KUKA KRL program: MyProgram_212().src

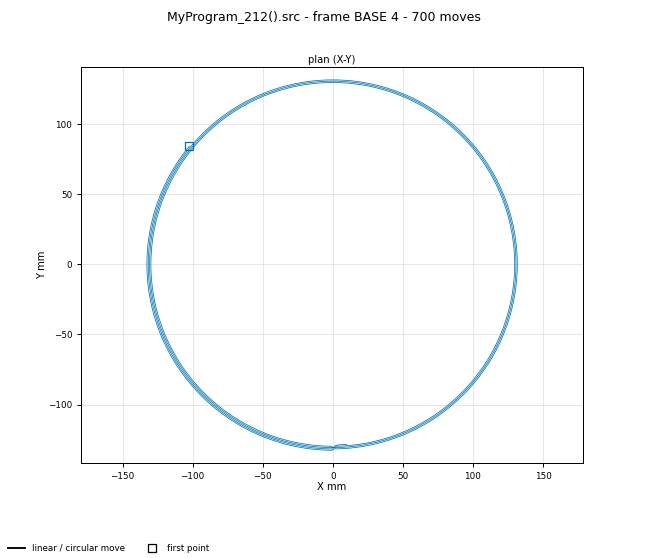
[picture p0: tool path of MyProgram_212().src in frame BASE 4, 700 of 700 moves have a stored position in this frame; points joined in program order, loops and branches not executed]
&ACCESS RVP
&REL 1
&PARAM TEMPLATE = C:\KRC\Roboter\Template\vorgabe
&PARAM EDITMASK = *
DEF MyProgram_212()
; ---- Setting reference (Base) ----
$BASE = BASE_DATA[4]

; --------------------------
; ---- Setting tool (TCP) ----
$TOOL = TOOL_DATA[3]
; --------------------------

$VEL.CP = VEL_APROX_PRINT
Startdeposition()
$VEL.CP = VEL_PRINT
LIN {X -102.2759,Y 84.4274,Z 150,A 136.9354,B 24.9526,C -1.5903,E1 24.8761,E2 309.4983} C_DIS
LIN {X -104.8003,Y 81.2724,Z 150,A 138.873,B 24.9523,C -1.5949,E1 24.8727,E2 307.5405} C_DIS
LIN {X -107.3516,Y 77.8713,Z 150,A 140.7222,B 24.9526,C -1.5904,E1 24.8697,E2 305.6931} C_DIS
LIN {X -109.8219,Y 74.3469,Z 150,A 142.615,B 24.9528,C -1.5868,E1 24.8667,E2 303.7996} C_DIS
LIN {X -112.2899,Y 70.5646,Z 150,A 144.5743,B 24.9531,C -1.5815,E1 24.8637,E2 301.8428} C_DIS
LIN {X -114.4855,Y 66.9437,Z 150,A 146.4163,B 24.9534,C -1.5768,E1 24.8611,E2 300.0027} C_DIS
LIN {X -116.5889,Y 63.2096,Z 150,A 148.3143,B 24.9536,C -1.5735,E1 24.8585,E2 298.1025} C_DIS
LIN {X -118.1366,Y 60.2624,Z 150,A 149.6641,B 24.9541,C -1.5649,E1 24.8568,E2 296.7661} C_DIS
LIN {X -120.6399,Y 55.0837,Z 150,A 152.138,B 24.9546,C -1.5567,E1 24.8539,E2 294.2982} C_DIS
LIN {X -122.2455,Y 51.4194,Z 150,A 153.8562,B 24.9549,C -1.5508,E1 24.852,E2 292.5846} C_DIS
LIN {X -123.5059,Y 48.3134,Z 150,A 155.3546,B 24.9551,C -1.5487,E1 24.8504,E2 291.0827} C_DIS
LIN {X -124.7525,Y 44.9959,Z 150,A 156.841,B 24.9555,C -1.5417,E1 24.849,E2 289.6046} C_DIS
LIN {X -125.7894,Y 42.0105,Z 150,A 158.2756,B 24.9555,C -1.5407,E1 24.8477,E2 288.1643} C_DIS
LIN {X -126.918,Y 38.468,Z 150,A 159.9592,B 24.9556,C -1.5393,E1 24.8463,E2 286.4744} C_DIS
LIN {X -128.0963,Y 34.3396,Z 150,A 161.7856,B 24.956,C -1.5319,E1 24.845,E2 284.655} C_DIS
LIN {X -129.0879,Y 30.4082,Z 150,A 163.4654,B 24.9566,C -1.5227,E1 24.8439,E2 282.9873} C_DIS
LIN {X -130.1134,Y 25.671,Z 150,A 165.7274,B 24.9565,C -1.5239,E1 24.8426,E2 280.709} C_DIS
LIN {X -130.8013,Y 21.8842,Z 150,A 167.3023,B 24.957,C -1.5143,E1 24.8418,E2 279.1478} C_DIS
LIN {X -131.3985,Y 17.9691,Z 150,A 169.2633,B 24.9567,C -1.5207,E1 24.841,E2 277.1597} C_DIS
LIN {X -131.9911,Y 12.8966,Z 150,A 171.2061,B 24.9578,C -1.5007,E1 24.8405,E2 275.2531} C_DIS
LIN {X -132.2828,Y 9.4461,Z 150,A 172.7501,B 24.958,C -1.498,E1 24.8401,E2 273.7061} C_DIS
LIN {X -132.5132,Y 5.3118,Z 150,A 174.5305,B 24.9583,C -1.4917,E1 24.8399,E2 271.93} C_DIS
LIN {X -132.6019,Y 2.1638,Z 150,A 175.9323,B 24.9585,C -1.4892,E1 24.8398,E2 270.5258} C_DIS
LIN {X -132.6079,Y -1.8067,Z 150,A 177.6767,B 24.9587,C -1.4849,E1 24.8398,E2 268.781} C_DIS
LIN {X -132.4992,Y -5.6705,Z 150,A 179.3978,B 24.9589,C -1.4819,E1 24.84,E2 267.0568} C_DIS
LIN {X -132.2762,Y -9.5365,Z 150,A -178.6096,B 24.9583,C -1.492,E1 24.8404,E2 265.0281} C_DIS
LIN {X -131.9496,Y -13.3288,Z 150,A -177.2383,B 24.9593,C -1.4733,E1 24.8408,E2 263.6932} C_DIS
LIN {X -131.5115,Y -17.1072,Z 150,A -175.6535,B 24.9598,C -1.4651,E1 24.8413,E2 262.1183} C_DIS
LIN {X -130.9322,Y -21.0996,Z 150,A -173.9674,B 24.9602,C -1.4567,E1 24.842,E2 260.4423} C_DIS
LIN {X -130.2084,Y -25.1739,Z 150,A -172.0506,B 24.9602,C -1.4573,E1 24.843,E2 258.5128} C_DIS
LIN {X -129.3647,Y -29.2021,Z 150,A -170.3174,B 24.9606,C -1.4494,E1 24.844,E2 256.7881} C_DIS
LIN {X -128.5771,Y -32.4932,Z 150,A -168.8558,B 24.9609,C -1.4448,E1 24.845,E2 255.3289} C_DIS
LIN {X -127.6515,Y -35.9585,Z 150,A -167.2711,B 24.9611,C -1.4417,E1 24.8461,E2 253.7426} C_DIS
LIN {X -126.4549,Y -39.9645,Z 150,A -165.4673,B 24.9614,C -1.436,E1 24.8476,E2 251.9419} C_DIS
LIN {X -125.4607,Y -42.9847,Z 150,A -164.0858,B 24.9616,C -1.4321,E1 24.8489,E2 250.5617} C_DIS
LIN {X -124.3657,Y -46.0568,Z 150,A -162.3318,B 24.9609,C -1.4448,E1 24.8506,E2 248.7676} C_DIS
LIN {X -123.1055,Y -49.3248,Z 150,A -161.0063,B 24.9616,C -1.431,E1 24.8519,E2 247.4675} C_DIS
LIN {X -121.3813,Y -53.4321,Z 150,A -159.1275,B 24.9621,C -1.4231,E1 24.854,E2 245.5972} C_DIS
LIN {X -119.781,Y -56.9243,Z 150,A -157.5495,B 24.9625,C -1.4143,E1 24.8558,E2 244.0315} C_DIS
LIN {X -118.2712,Y -59.998,Z 150,A -156.0681,B 24.9627,C -1.4102,E1 24.8577,E2 242.5519} C_DIS
LIN {X -116.633,Y -63.1286,Z 150,A -154.4098,B 24.9627,C -1.4123,E1 24.8599,E2 240.8797} C_DIS
LIN {X -114.4561,Y -66.9937,Z 150,A -152.521,B 24.963,C -1.4057,E1 24.8625,E2 238.997} C_DIS
LIN {X -112.2679,Y -70.5995,Z 150,A -150.6806,B 24.9632,C -1.4017,E1 24.8652,E2 237.1567} C_DIS
LIN {X -109.8561,Y -74.2964,Z 150,A -149.0433,B 24.9642,C -1.3834,E1 24.8677,E2 235.5548} C_DIS
LIN {X -108.2088,Y -76.6762,Z 150,A -147.5106,B 24.9636,C -1.3941,E1 24.8702,E2 233.9891} C_DIS
LIN {X -105.6102,Y -80.2182,Z 150,A -145.571,B 24.9637,C -1.3914,E1 24.8734,E2 232.0466} C_DIS
LIN {X -102.8564,Y -83.7194,Z 150,A -143.6381,B 24.964,C -1.3871,E1 24.8768,E2 230.1148} C_DIS
LIN {X -99.9263,Y -87.1954,Z 150,A -141.6922,B 24.9642,C -1.3816,E1 24.8803,E2 228.1732} C_DIS
LIN {X -96.9225,Y -90.5228,Z 150,A -139.7451,B 24.9644,C -1.3777,E1 24.884,E2 226.2267} C_DIS
LIN {X -93.8055,Y -93.7496,Z 150,A -137.7952,B 24.9646,C -1.374,E1 24.8878,E2 224.2774} C_DIS
LIN {X -90.7475,Y -96.7126,Z 150,A -135.9208,B 24.9647,C -1.3718,E1 24.8916,E2 222.4003} C_DIS
LIN {X -87.5016,Y -99.6591,Z 150,A -134.0241,B 24.9649,C -1.3681,E1 24.8956,E2 220.5048} C_DIS
LIN {X -84.1587,Y -102.4974,Z 150,A -132.1382,B 24.9651,C -1.364,E1 24.8996,E2 218.6215} C_DIS
LIN {X -80.768,Y -105.1898,Z 150,A -130.2526,B 24.9653,C -1.3613,E1 24.9038,E2 216.7355} C_DIS
LIN {X -77.1748,Y -107.8534,Z 150,A -128.3209,B 24.9655,C -1.3579,E1 24.9081,E2 214.8051} C_DIS
LIN {X -73.3393,Y -110.4979,Z 150,A -126.2967,B 24.9656,C -1.3551,E1 24.9128,E2 212.7807} C_DIS
LIN {X -69.7226,Y -112.8151,Z 150,A -124.4068,B 24.9656,C -1.3539,E1 24.9173,E2 210.8876} C_DIS
LIN {X -65.5266,Y -115.3023,Z 150,A -122.009,B 24.9651,C -1.3657,E1 24.9232,E2 208.4548} C_DIS
LIN {X -62.1909,Y -117.1343,Z 150,A -120.678,B 24.966,C -1.3475,E1 24.9264,E2 207.1634} C_DIS
LIN {X -58.8187,Y -118.8621,Z 150,A -119.1574,B 24.9664,C -1.3395,E1 24.9301,E2 205.6577} C_DIS
LIN {X -55.5234,Y -120.4366,Z 150,A -117.5891,B 24.9665,C -1.3371,E1 24.9341,E2 204.0912} C_DIS
LIN {X -52.7823,Y -121.6629,Z 150,A -116.3412,B 24.9667,C -1.3331,E1 24.9373,E2 202.8497} C_DIS
LIN {X -49.8052,Y -122.9118,Z 150,A -114.8731,B 24.9666,C -1.3354,E1 24.9411,E2 201.3728} C_DIS
LIN {X -46.6232,Y -124.1536,Z 150,A -113.396,B 24.9666,C -1.334,E1 24.9449,E2 199.8959} C_DIS
LIN {X -43.6406,Y -125.2333,Z 150,A -111.9841,B 24.9666,C -1.3349,E1 24.9486,E2 198.479} C_DIS
LIN {X -40.3714,Y -126.3249,Z 150,A -110.5705,B 24.9669,C -1.3299,E1 24.9524,E2 197.0749} C_DIS
LIN {X -36.267,Y -127.5652,Z 150,A -108.6068,B 24.9667,C -1.3343,E1 24.9577,E2 195.0975} C_DIS
LIN {X -32.2664,Y -128.6346,Z 150,A -106.7479,B 24.9665,C -1.3368,E1 24.9627,E2 193.2298} C_DIS
LIN {X -28.2908,Y -129.567,Z 150,A -105.0688,B 24.9668,C -1.3315,E1 24.9673,E2 191.5612} C_DIS
LIN {X -24.1984,Y -130.3949,Z 150,A -103.1867,B 24.9666,C -1.3348,E1 24.9724,E2 189.6691} C_DIS
LIN {X -20.4691,Y -131.0303,Z 150,A -101.6331,B 24.9669,C -1.3302,E1 24.9767,E2 188.1251} C_DIS
LIN {X -16.8245,Y -131.5485,Z 150,A -99.9382,B 24.9666,C -1.3353,E1 24.9814,E2 186.4168} C_DIS
LIN {X -13.0464,Y -131.9767,Z 150,A -98.3401,B 24.9667,C -1.3328,E1 24.9859,E2 184.8237} C_DIS
LIN {X -8.7557,Y -132.3315,Z 150,A -96.4662,B 24.9667,C -1.3334,E1 24.9911,E2 182.9475} C_DIS
LIN {X -4.8645,Y -132.5306,Z 150,A -94.7842,B 24.9667,C -1.3335,E1 24.9958,E2 181.2649} C_DIS
LIN {X -0.6926,Y -132.6178,Z 150,A -93.0498,B 24.9669,C -1.3303,E1 25.0006,E2 179.5381} C_DIS
LIN {X -0.6926,Y -132.6178,Z 150,A -93.0498,B 24.9669,C -1.3303,E1 25.0006,E2 179.5381} C_DIS
Enddeposition()
LIN {X 0.9332,Y -131.667,Z 150,A -92.4211,B 24.2531,C -1.1938,E1 24.2824,E2 179.1428} C_DIS
Startdeposition()
$VEL.CP = VEL_PRINT
LIN {X -0.8148,Y -131.6701,Z 150,A -93.6093,B 24.2541,C -1.1721,E1 24.279,E2 180.3838} C_DIS
LIN {X -4.9682,Y -131.5789,Z 150,A -95.3944,B 24.2541,C -1.173,E1 24.274,E2 182.1669} C_DIS
LIN {X -8.4532,Y -131.4014,Z 150,A -96.8971,B 24.2541,C -1.1737,E1 24.2698,E2 183.6683} C_DIS
LIN {X -11.7251,Y -131.151,Z 150,A -98.299,B 24.2541,C -1.1751,E1 24.2659,E2 185.0676} C_DIS
LIN {X -15.4301,Y -130.7653,Z 150,A -99.9452,B 24.2541,C -1.174,E1 24.2613,E2 186.7174} C_DIS
LIN {X -18.6917,Y -130.339,Z 150,A -101.3801,B 24.2541,C -1.1742,E1 24.2574,E2 188.1531} C_DIS
LIN {X -22.0826,Y -129.8081,Z 150,A -102.8712,B 24.2541,C -1.1747,E1 24.2532,E2 189.6442} C_DIS
LIN {X -25.4894,Y -129.184,Z 150,A -104.363,B 24.254,C -1.1761,E1 24.2492,E2 191.1344} C_DIS
LIN {X -27.9438,Y -128.6731,Z 150,A -105.4714,B 24.254,C -1.1757,E1 24.2461,E2 192.245} C_DIS
LIN {X -31.6236,Y -127.8208,Z 150,A -107.1045,B 24.254,C -1.1771,E1 24.2417,E2 193.877} C_DIS
LIN {X -34.5863,Y -127.0505,Z 150,A -108.4405,B 24.2539,C -1.1777,E1 24.2381,E2 195.2135} C_DIS
LIN {X -37.6577,Y -126.1742,Z 150,A -109.8155,B 24.2539,C -1.1794,E1 24.2344,E2 196.5867} C_DIS
LIN {X -40.1695,Y -125.3953,Z 150,A -110.9923,B 24.2539,C -1.1788,E1 24.2313,E2 197.7674} C_DIS
LIN {X -43.3579,Y -124.329,Z 150,A -112.4851,B 24.2539,C -1.1785,E1 24.2273,E2 199.2636} C_DIS
LIN {X -46.6138,Y -123.1459,Z 150,A -113.9587,B 24.2537,C -1.1816,E1 24.2235,E2 200.733} C_DIS
LIN {X -49.5228,Y -122.0046,Z 150,A -115.3569,B 24.2537,C -1.1811,E1 24.2198,E2 202.1355} C_DIS
LIN {X -52.7628,Y -120.6397,Z 150,A -116.8575,B 24.2536,C -1.1842,E1 24.216,E2 203.6323} C_DIS
LIN {X -56.0138,Y -119.1665,Z 150,A -118.4198,B 24.2536,C -1.1855,E1 24.212,E2 205.1953} C_DIS
LIN {X -58.9958,Y -117.7187,Z 150,A -119.9107,B 24.2536,C -1.185,E1 24.2083,E2 206.6915} C_DIS
LIN {X -62.6349,Y -115.8233,Z 150,A -121.6598,B 24.2534,C -1.1891,E1 24.204,E2 208.4356} C_DIS
LIN {X -65.5557,Y -114.1955,Z 150,A -123.2346,B 24.2535,C -1.1854,E1 24.2001,E2 210.0242} C_DIS
LIN {X -69.2621,Y -111.9863,Z 150,A -125.1463,B 24.2535,C -1.1866,E1 24.1955,E2 211.9391} C_DIS
LIN {X -72.6874,Y -109.7938,Z 150,A -126.8783,B 24.2533,C -1.1912,E1 24.1915,E2 213.6656} C_DIS
LIN {X -76.2415,Y -107.3566,Z 150,A -128.6594,B 24.2529,C -1.1989,E1 24.1874,E2 215.4341} C_DIS
LIN {X -79.3271,Y -105.0963,Z 150,A -130.393,B 24.2529,C -1.1986,E1 24.1835,E2 217.175} C_DIS
LIN {X -82.6146,Y -102.5322,Z 150,A -132.2309,B 24.2529,C -1.2008,E1 24.1795,E2 219.0145} C_DIS
LIN {X -85.8963,Y -99.7991,Z 150,A -134.0859,B 24.2526,C -1.2046,E1 24.1756,E2 220.8676} C_DIS
LIN {X -88.9982,Y -97.0431,Z 150,A -135.9311,B 24.2526,C -1.2064,E1 24.1717,E2 222.7161} C_DIS
LIN {X -91.8951,Y -94.3054,Z 150,A -137.5823,B 24.2522,C -1.214,E1 24.1684,E2 224.3558} C_DIS
LIN {X -94.2367,Y -91.9651,Z 150,A -139.1194,B 24.2522,C -1.2125,E1 24.1654,E2 225.9031} C_DIS
LIN {X -97.2286,Y -88.7965,Z 150,A -140.9291,B 24.2519,C -1.2209,E1 24.162,E2 227.7007} C_DIS
LIN {X -99.4528,Y -86.2977,Z 150,A -142.3879,B 24.2517,C -1.2241,E1 24.1593,E2 229.1584} C_DIS
LIN {X -101.8838,Y -83.413,Z 150,A -144.1386,B 24.2517,C -1.2229,E1 24.1561,E2 230.9203} C_DIS
LIN {X -104.5752,Y -80.0129,Z 150,A -146.0156,B 24.2515,C -1.228,E1 24.1529,E2 232.7941} C_DIS
LIN {X -107.0701,Y -76.6422,Z 150,A -147.8508,B 24.2513,C -1.2321,E1 24.1499,E2 234.6284} C_DIS
LIN {X -109.4269,Y -73.2379,Z 150,A -149.6804,B 24.2512,C -1.2355,E1 24.147,E2 236.4593} C_DIS
LIN {X -111.5415,Y -69.9761,Z 150,A -151.3797,B 24.251,C -1.2396,E1 24.1445,E2 238.1574} C_DIS
LIN {X -113.7761,Y -66.2809,Z 150,A -153.3185,B 24.2509,C -1.2419,E1 24.1417,E2 240.1008} C_DIS
LIN {X -115.7952,Y -62.6871,Z 150,A -155.1261,B 24.2507,C -1.2462,E1 24.1393,E2 241.9078} C_DIS
LIN {X -117.5957,Y -59.2374,Z 150,A -156.678,B 24.2501,C -1.2575,E1 24.1373,E2 243.4405} C_DIS
LIN {X -118.9999,Y -56.3627,Z 150,A -158.0771,B 24.2499,C -1.2612,E1 24.1356,E2 244.8385} C_DIS
LIN {X -120.5329,Y -53.0096,Z 150,A -159.6961,B 24.2498,C -1.2651,E1 24.1338,E2 246.457} C_DIS
LIN {X -121.8177,Y -49.9865,Z 150,A -161.133,B 24.2496,C -1.269,E1 24.1322,E2 247.8927} C_DIS
LIN {X -123.0209,Y -46.9474,Z 150,A -162.5629,B 24.2494,C -1.2729,E1 24.1308,E2 249.3214} C_DIS
LIN {X -123.9898,Y -44.3194,Z 150,A -163.8263,B 24.2493,C -1.2745,E1 24.1296,E2 250.5881} C_DIS
LIN {X -125.0082,Y -41.3591,Z 150,A -165.1834,B 24.2491,C -1.2789,E1 24.1284,E2 251.9425} C_DIS
LIN {X -126.0115,Y -38.1942,Z 150,A -166.5921,B 24.2488,C -1.285,E1 24.1272,E2 253.3447} C_DIS
LIN {X -126.826,Y -35.3942,Z 150,A -167.883,B 24.2486,C -1.2879,E1 24.1262,E2 254.6362} C_DIS
LIN {X -127.6413,Y -32.3308,Z 150,A -169.2828,B 24.2485,C -1.2912,E1 24.1252,E2 256.0363} C_DIS
LIN {X -128.4131,Y -29.1152,Z 150,A -170.728,B 24.2482,C -1.2955,E1 24.1243,E2 257.4798} C_DIS
LIN {X -129.0911,Y -25.9459,Z 150,A -172.1707,B 24.2481,C -1.2984,E1 24.1235,E2 258.924} C_DIS
LIN {X -129.7497,Y -22.4326,Z 150,A -173.7009,B 24.2478,C -1.3045,E1 24.1227,E2 260.4487} C_DIS
LIN {X -130.2397,Y -19.3862,Z 150,A -175.0507,B 24.2476,C -1.3085,E1 24.1222,E2 261.7971} C_DIS
LIN {X -130.6553,Y -16.3526,Z 150,A -176.3905,B 24.2474,C -1.3124,E1 24.1217,E2 263.1355} C_DIS
LIN {X -130.9862,Y -13.4413,Z 150,A -177.6717,B 24.2472,C -1.3163,E1 24.1213,E2 264.4153} C_DIS
LIN {X -131.2685,Y -10.3335,Z 150,A -179.0367,B 24.247,C -1.3203,E1 24.121,E2 265.7788} C_DIS
LIN {X -131.4334,Y -7.9342,Z 150,A 179.8473,B 24.247,C -1.3206,E1 24.1208,E2 266.9011} C_DIS
LIN {X -131.5972,Y -4.4983,Z 150,A 178.404,B 24.2466,C -1.3279,E1 24.1206,E2 268.3355} C_DIS
LIN {X -131.6648,Y -1.5621,Z 150,A 177.1632,B 24.2463,C -1.3338,E1 24.1206,E2 269.5697} C_DIS
LIN {X -131.6678,Y 1.287,Z 150,A 175.8565,B 24.2463,C -1.3348,E1 24.1206,E2 270.882} C_DIS
LIN {X -131.5674,Y 5.2629,Z 150,A 174.0649,B 24.2461,C -1.3377,E1 24.1206,E2 272.6777} C_DIS
LIN {X -131.3775,Y 8.8404,Z 150,A 172.5524,B 24.2457,C -1.3449,E1 24.1209,E2 274.182} C_DIS
LIN {X -131.151,Y 11.7251,Z 150,A 171.279,B 24.2455,C -1.3484,E1 24.1212,E2 275.4547} C_DIS
LIN {X -130.836,Y 14.837,Z 150,A 169.9092,B 24.2453,C -1.3524,E1 24.1217,E2 276.8231} C_DIS
LIN {X -130.4708,Y 17.76,Z 150,A 168.6347,B 24.2451,C -1.3569,E1 24.1221,E2 278.0944} C_DIS
LIN {X -130.0208,Y 20.7999,Z 150,A 167.2633,B 24.2449,C -1.3597,E1 24.1227,E2 279.4673} C_DIS
LIN {X -129.4958,Y 23.8514,Z 150,A 165.9042,B 24.2447,C -1.3636,E1 24.1234,E2 280.8253} C_DIS
LIN {X -128.9359,Y 26.7086,Z 150,A 164.6144,B 24.2446,C -1.3667,E1 24.1241,E2 282.1154} C_DIS
LIN {X -128.2739,Y 29.725,Z 150,A 163.2857,B 24.2443,C -1.3717,E1 24.1249,E2 283.4399} C_DIS
LIN {X -127.4587,Y 33.0503,Z 150,A 161.771,B 24.2441,C -1.3754,E1 24.1259,E2 284.9548} C_DIS
LIN {X -126.7683,Y 35.6006,Z 150,A 160.5988,B 24.244,C -1.3781,E1 24.1268,E2 286.1274} C_DIS
LIN {X -125.8001,Y 38.8849,Z 150,A 159.1337,B 24.2437,C -1.3839,E1 24.128,E2 287.5869} C_DIS
LIN {X -124.8443,Y 41.8511,Z 150,A 157.7294,B 24.2435,C -1.386,E1 24.1292,E2 288.9944} C_DIS
LIN {X -123.7058,Y 45.1071,Z 150,A 156.251,B 24.2432,C -1.3918,E1 24.1306,E2 290.4673} C_DIS
LIN {X -122.5781,Y 48.0866,Z 150,A 154.8065,B 24.2432,C -1.3935,E1 24.132,E2 291.9161} C_DIS
LIN {X -121.3681,Y 51.0632,Z 150,A 153.3887,B 24.243,C -1.3969,E1 24.1335,E2 293.3336} C_DIS
LIN {X -119.9077,Y 54.4074,Z 150,A 151.8353,B 24.2426,C -1.4033,E1 24.1353,E2 294.8801} C_DIS
LIN {X -118.4528,Y 57.5078,Z 150,A 150.3202,B 24.2424,C -1.4067,E1 24.1371,E2 296.3955} C_DIS
LIN {X -116.9645,Y 60.4774,Z 150,A 148.8639,B 24.2422,C -1.4106,E1 24.1389,E2 297.8504} C_DIS
LIN {X -115.4701,Y 63.2831,Z 150,A 147.3765,B 24.2422,C -1.4099,E1 24.1409,E2 299.3476} C_DIS
LIN {X -113.3517,Y 67.0041,Z 150,A 145.5412,B 24.2419,C -1.4166,E1 24.1435,E2 301.1762} C_DIS
LIN {X -111.1242,Y 70.6373,Z 150,A 143.7265,B 24.2415,C -1.4238,E1 24.1462,E2 302.9829} C_DIS
LIN {X -109.312,Y 73.4102,Z 150,A 142.2732,B 24.2413,C -1.4273,E1 24.1484,E2 304.4352} C_DIS
LIN {X -107.047,Y 76.6745,Z 150,A 140.4571,B 24.2413,C -1.4281,E1 24.1513,E2 306.2584} C_DIS
LIN {X -104.3697,Y 80.2816,Z 150,A 138.5679,B 24.2408,C -1.4365,E1 24.1545,E2 308.1366} C_DIS
LIN {X -102.226,Y 82.9943,Z 150,A 137.0243,B 24.2407,C -1.4387,E1 24.1572,E2 309.6823} C_DIS
LIN {X -99.5321,Y 86.2063,Z 150,A 135.2124,B 24.2404,C -1.4441,E1 24.1605,E2 311.4896} C_DIS
LIN {X -97.2692,Y 88.7516,Z 150,A 133.7284,B 24.2401,C -1.4478,E1 24.1632,E2 312.9714} C_DIS
LIN {X -94.9399,Y 91.2391,Z 150,A 132.2136,B 24.2401,C -1.45,E1 24.1661,E2 314.4875} C_DIS
LIN {X -92.0249,Y 94.178,Z 150,A 130.3391,B 24.24,C -1.451,E1 24.1699,E2 316.3677} C_DIS
LIN {X -88.7965,Y 97.2286,Z 150,A 128.4899,B 24.2395,C -1.4595,E1 24.1736,E2 318.204} C_DIS
LIN {X -86.2977,Y 99.4528,Z 150,A 127.021,B 24.2393,C -1.4622,E1 24.1767,E2 319.6722} C_DIS
LIN {X -83.6525,Y 101.6881,Z 150,A 125.4423,B 24.2393,C -1.4622,E1 24.1801,E2 321.257} C_DIS
LIN {X -80.3295,Y 104.333,Z 150,A 123.6507,B 24.239,C -1.4689,E1 24.184,E2 323.0393} C_DIS
LIN {X -77.6643,Y 106.3317,Z 150,A 122.1885,B 24.2388,C -1.4713,E1 24.1873,E2 324.5008} C_DIS
LIN {X -74.8561,Y 108.3271,Z 150,A 120.5702,B 24.239,C -1.4688,E1 24.191,E2 326.131} C_DIS
LIN {X -71.3969,Y 110.6374,Z 150,A 118.7929,B 24.2387,C -1.4739,E1 24.1952,E2 327.9019} C_DIS
LIN {X -67.8273,Y 112.861,Z 150,A 117.0305,B 24.2383,C -1.4805,E1 24.1993,E2 329.6539} C_DIS
LIN {X -64.4639,Y 114.8148,Z 150,A 115.2856,B 24.2383,C -1.4811,E1 24.2036,E2 331.4027} C_DIS
LIN {X -60.7251,Y 116.8344,Z 150,A 113.4927,B 24.2379,C -1.4869,E1 24.208,E2 333.1866} C_DIS
LIN {X -57.6492,Y 118.383,Z 150,A 111.9816,B 24.2379,C -1.4887,E1 24.2117,E2 334.6973} C_DIS
LIN {X -54.6208,Y 119.8106,Z 150,A 110.5189,B 24.2377,C -1.4907,E1 24.2154,E2 336.1589} C_DIS
LIN {X -51.6849,Y 121.1057,Z 150,A 109.114,B 24.2377,C -1.4923,E1 24.219,E2 337.5632} C_DIS
LIN {X -49.0101,Y 122.2113,Z 150,A 107.8485,B 24.2375,C -1.4938,E1 24.2223,E2 338.8279} C_DIS
LIN {X -45.8227,Y 123.4422,Z 150,A 106.3368,B 24.2375,C -1.4946,E1 24.2263,E2 340.3409} C_DIS
LIN {X -42.3661,Y 124.6728,Z 150,A 104.7722,B 24.2373,C -1.4981,E1 24.2304,E2 341.9002} C_DIS
LIN {X -39.4102,Y 125.6379,Z 150,A 103.4268,B 24.2372,C -1.5001,E1 24.2339,E2 343.2433} C_DIS
LIN {X -36.4873,Y 126.5169,Z 150,A 102.0875,B 24.2372,C -1.5011,E1 24.2375,E2 344.5825} C_DIS
LIN {X -33.4291,Y 127.3591,Z 150,A 100.6904,B 24.2371,C -1.5017,E1 24.2413,E2 345.9803} C_DIS
LIN {X -30.1974,Y 128.1646,Z 150,A 99.2568,B 24.2369,C -1.5038,E1 24.2452,E2 347.4108} C_DIS
LIN {X -27.4225,Y 128.7856,Z 150,A 97.9934,B 24.2369,C -1.5037,E1 24.2486,E2 348.6762} C_DIS
LIN {X -24.0686,Y 129.4556,Z 150,A 96.5273,B 24.2369,C -1.5059,E1 24.2526,E2 350.1384} C_DIS
LIN {X -21.0163,Y 129.986,Z 150,A 95.1792,B 24.2368,C -1.5069,E1 24.2564,E2 351.4855} C_DIS
LIN {X -18.3702,Y 130.3849,Z 150,A 93.9694,B 24.2368,C -1.5055,E1 24.2597,E2 352.6998} C_DIS
LIN {X -14.0764,Y 130.9179,Z 150,A 92.0983,B 24.2368,C -1.5071,E1 24.2649,E2 354.5681} C_DIS
LIN {X -10.8669,Y 131.2235,Z 150,A 90.6889,B 24.2368,C -1.5075,E1 24.2688,E2 355.9774} C_DIS
LIN {X -7.4582,Y 131.4627,Z 150,A 89.2712,B 24.2365,C -1.5114,E1 24.2727,E2 357.386} C_DIS
LIN {X -2.9226,Y 131.6422,Z 150,A 87.1562,B 24.2369,C -1.5052,E1 24.2787,E2 359.5166} C_DIS
LIN {X 0.7468,Y 131.6705,Z 150,A 85.6682,B 24.2365,C -1.5108,E1 24.2828,E2 360.9907} C_DIS
LIN {X 3.7909,Y 131.6181,Z 150,A 84.3302,B 24.2365,C -1.5103,E1 24.2865,E2 362.3297} C_DIS
LIN {X 7.2472,Y 131.4745,Z 150,A 82.8404,B 24.2365,C -1.5111,E1 24.2907,E2 363.8171} C_DIS
LIN {X 10.3335,Y 131.2685,Z 150,A 81.3369,B 24.237,C -1.5033,E1 24.2949,E2 365.3388} C_DIS
LIN {X 13.9989,Y 130.9262,Z 150,A 79.8614,B 24.2366,C -1.5093,E1 24.299,E2 366.7987} C_DIS
LIN {X 17.2091,Y 130.543,Z 150,A 78.4643,B 24.2366,C -1.5095,E1 24.3028,E2 368.1942} C_DIS
LIN {X 20.7999,Y 130.0208,Z 150,A 76.8983,B 24.2366,C -1.5096,E1 24.3072,E2 369.7585} C_DIS
LIN {X 23.8514,Y 129.4958,Z 150,A 75.5742,B 24.2366,C -1.5102,E1 24.3108,E2 371.0795} C_DIS
LIN {X 26.6183,Y 128.9542,Z 150,A 74.2994,B 24.2367,C -1.5073,E1 24.3143,E2 372.3598} C_DIS
LIN {X 30.0883,Y 128.1909,Z 150,A 72.7788,B 24.2367,C -1.5077,E1 24.3184,E2 373.8773} C_DIS
LIN {X 33.0503,Y 127.4587,Z 150,A 71.4507,B 24.2367,C -1.5069,E1 24.322,E2 375.2054} C_DIS
LIN {X 35.5851,Y 126.7726,Z 150,A 70.2936,B 24.2368,C -1.5054,E1 24.3251,E2 376.3641} C_DIS
LIN {X 38.7752,Y 125.8337,Z 150,A 68.841,B 24.2369,C -1.504,E1 24.329,E2 377.8174} C_DIS
LIN {X 41.9333,Y 124.817,Z 150,A 67.4256,B 24.2369,C -1.5042,E1 24.3328,E2 379.2296} C_DIS
LIN {X 44.8971,Y 123.7815,Z 150,A 66.018,B 24.2371,C -1.5009,E1 24.3365,E2 380.6423} C_DIS
LIN {X 48.3607,Y 122.4715,Z 150,A 64.4507,B 24.2371,C -1.5015,E1 24.3406,E2 382.2047} C_DIS
LIN {X 51.1418,Y 121.3352,Z 150,A 63.1165,B 24.2372,C -1.4987,E1 24.344,E2 383.5424} C_DIS
LIN {X 54.4074,Y 119.9077,Z 150,A 61.5864,B 24.2372,C -1.4979,E1 24.3479,E2 385.0705} C_DIS
LIN {X 57.5078,Y 118.4528,Z 150,A 60.1018,B 24.2374,C -1.4964,E1 24.3517,E2 386.5549} C_DIS
LIN {X 60.4774,Y 116.9645,Z 150,A 58.6592,B 24.2374,C -1.4946,E1 24.3552,E2 387.9976} C_DIS
LIN {X 63.4201,Y 115.3954,Z 150,A 57.1151,B 24.2379,C -1.4879,E1 24.3591,E2 389.5536} C_DIS
LIN {X 67.1066,Y 113.291,Z 150,A 55.2291,B 24.2381,C -1.4832,E1 24.3636,E2 391.445} C_DIS
LIN {X 71.0707,Y 110.8467,Z 150,A 53.2627,B 24.2381,C -1.483,E1 24.3683,E2 393.4052} C_DIS
LIN {X 74.8066,Y 108.3611,Z 150,A 51.3945,B 24.2381,C -1.4841,E1 24.3726,E2 395.2644} C_DIS
LIN {X 78.1267,Y 105.992,Z 150,A 49.5798,B 24.2384,C -1.4789,E1 24.3767,E2 397.0851} C_DIS
LIN {X 81.5864,Y 103.3527,Z 150,A 47.6774,B 24.2386,C -1.4749,E1 24.3809,E2 398.9899} C_DIS
LIN {X 84.9128,Y 100.6379,Z 150,A 45.8269,B 24.2388,C -1.4722,E1 24.3849,E2 400.8397} C_DIS
LIN {X 88.1538,Y 97.8115,Z 150,A 44.0258,B 24.2388,C -1.472,E1 24.3886,E2 402.6338} C_DIS
LIN {X 90.6228,Y 95.5284,Z 150,A 42.5203,B 24.2391,C -1.4668,E1 24.3917,E2 404.1457} C_DIS
LIN {X 93.6307,Y 92.582,Z 150,A 40.6405,B 24.2394,C -1.4603,E1 24.3954,E2 406.0329} C_DIS
LIN {X 96.6521,Y 89.4236,Z 150,A 38.8513,B 24.2394,C -1.4619,E1 24.3988,E2 407.8103} C_DIS
LIN {X 99.0232,Y 86.79,Z 150,A 37.1921,B 24.2399,C -1.4522,E1 24.402,E2 409.4852} C_DIS
LIN {X 101.6881,Y 83.6525,Z 150,A 35.5388,B 24.2397,C -1.4551,E1 24.4049,E2 411.1238} C_DIS
LIN {X 103.85,Y 80.9527,Z 150,A 33.9006,B 24.2403,C -1.4445,E1 24.4078,E2 412.7797} C_DIS
LIN {X 106.5108,Y 77.4178,Z 150,A 32.0259,B 24.2405,C -1.4423,E1 24.4109,E2 414.6504} C_DIS
LIN {X 109.002,Y 73.8688,Z 150,A 30.1667,B 24.2406,C -1.4388,E1 24.4138,E2 416.5086} C_DIS
LIN {X 111.4021,Y 70.1969,Z 150,A 28.2614,B 24.2409,C -1.4339,E1 24.4167,E2 418.4158} C_DIS
LIN {X 113.6885,Y 66.4308,Z 150,A 26.3696,B 24.2411,C -1.4301,E1 24.4194,E2 420.307} C_DIS
LIN {X 115.7952,Y 62.6871,Z 150,A 24.4498,B 24.2416,C -1.4222,E1 24.422,E2 422.2354} C_DIS
LIN {X 117.6652,Y 59.1011,Z 150,A 22.8411,B 24.2414,C -1.4252,E1 24.424,E2 423.8282} C_DIS
LIN {X 118.9646,Y 56.4365,Z 150,A 21.5702,B 24.2416,C -1.4225,E1 24.4256,E2 425.0985} C_DIS
LIN {X 120.3008,Y 53.5285,Z 150,A 20.1573,B 24.2418,C -1.4174,E1 24.4272,E2 426.5158} C_DIS
LIN {X 121.8177,Y 49.9865,Z 150,A 18.5135,B 24.242,C -1.4141,E1 24.429,E2 428.1581} C_DIS
LIN {X 122.8822,Y 47.3043,Z 150,A 17.2702,B 24.2422,C -1.4111,E1 24.4302,E2 429.4017} C_DIS
LIN {X 124.0316,Y 44.2035,Z 150,A 15.8401,B 24.2424,C -1.4072,E1 24.4316,E2 430.833} C_DIS
LIN {X 125.0757,Y 41.1564,Z 150,A 14.4458,B 24.2426,C -1.4033,E1 24.4328,E2 432.2285} C_DIS
LIN {X 126.0584,Y 38.0408,Z 150,A 13.022,B 24.2428,C -1.3988,E1 24.434,E2 433.6549} C_DIS
LIN {X 126.8771,Y 35.2113,Z 150,A 11.7156,B 24.2431,C -1.3936,E1 24.435,E2 434.9662} C_DIS
LIN {X 127.8208,Y 31.6236,Z 150,A 10.166,B 24.2432,C -1.3919,E1 24.4361,E2 436.5106} C_DIS
LIN {X 128.4634,Y 28.8953,Z 150,A 8.9321,B 24.2435,C -1.3873,E1 24.4369,E2 437.7482} C_DIS
LIN {X 129.1618,Y 25.5982,Z 150,A 7.5025,B 24.2436,C -1.3846,E1 24.4377,E2 439.1758} C_DIS
LIN {X 129.8823,Y 21.6376,Z 150,A 5.7376,B 24.244,C -1.3783,E1 24.4385,E2 440.9451} C_DIS
LIN {X 130.414,Y 18.1664,Z 150,A 4.2319,B 24.2442,C -1.3746,E1 24.4391,E2 442.4507} C_DIS
LIN {X 130.8355,Y 14.8414,Z 150,A 2.8052,B 24.2443,C -1.3715,E1 24.4396,E2 443.8762} C_DIS
LIN {X 131.1213,Y 12.0467,Z 150,A 1.6317,B 24.2443,C -1.3702,E1 24.4399,E2 445.0458} C_DIS
LIN {X 131.3418,Y 9.3298,Z 150,A 0.3718,B 24.2448,C -1.3624,E1 24.4402,E2 446.3168} C_DIS
LIN {X 131.5676,Y 5.2573,Z 150,A -1.3925,B 24.2451,C -1.3572,E1 24.4404,E2 448.0829} C_DIS
LIN {X 131.6648,Y 1.5621,Z 150,A -2.8946,B 24.2451,C -1.3575,E1 24.4405,E2 449.575} C_DIS
LIN {X 131.6578,Y -1.9827,Z 150,A -4.5136,B 24.2455,C -1.3484,E1 24.4405,E2 451.2061} C_DIS
LIN {X 131.565,Y -5.3254,Z 150,A -5.9415,B 24.2457,C -1.3451,E1 24.4404,E2 452.6332} C_DIS
LIN {X 131.3775,Y -8.8404,Z 150,A -7.44,B 24.2459,C -1.3418,E1 24.4401,E2 454.1306} C_DIS
LIN {X 131.1836,Y -11.3386,Z 150,A -8.5723,B 24.2462,C -1.336,E1 24.4398,E2 455.2698} C_DIS
LIN {X 130.8742,Y -14.4817,Z 150,A -9.8655,B 24.2462,C -1.3358,E1 24.4395,E2 456.5557} C_DIS
LIN {X 130.527,Y -17.3317,Z 150,A -11.1371,B 24.2465,C -1.3305,E1 24.439,E2 457.8323} C_DIS
LIN {X 130.0716,Y -20.4719,Z 150,A -12.5158,B 24.2467,C -1.3261,E1 24.4384,E2 459.2133} C_DIS
LIN {X 129.5225,Y -23.7022,Z 150,A -13.9405,B 24.2469,C -1.3214,E1 24.4378,E2 460.6406} C_DIS
LIN {X 128.8723,Y -27.0209,Z 150,A -15.3889,B 24.2471,C -1.3179,E1 24.437,E2 462.0889} C_DIS
LIN {X 128.1909,Y -30.0883,Z 150,A -16.7489,B 24.2473,C -1.3138,E1 24.4361,E2 463.4506} C_DIS
LIN {X 127.4587,Y -33.0503,Z 150,A -18.0696,B 24.2475,C -1.3099,E1 24.4352,E2 464.7728} C_DIS
LIN {X 126.6224,Y -36.1222,Z 150,A -19.4472,B 24.2477,C -1.3058,E1 24.4342,E2 466.1521} C_DIS
LIN {X 125.6727,Y -39.3013,Z 150,A -20.8829,B 24.2479,C -1.3016,E1 24.433,E2 467.5895} C_DIS
LIN {X 124.8553,Y -41.8181,Z 150,A -22.0329,B 24.2481,C -1.2981,E1 24.432,E2 468.7414} C_DIS
LIN {X 123.7784,Y -44.9056,Z 150,A -23.488,B 24.2484,C -1.2919,E1 24.4306,E2 470.2031} C_DIS
LIN {X 122.4715,Y -48.3607,Z 150,A -25.0286,B 24.2485,C -1.2903,E1 24.4291,E2 471.7386} C_DIS
LIN {X 121.4186,Y -50.9422,Z 150,A -26.2586,B 24.2487,C -1.2857,E1 24.4278,E2 472.9729} C_DIS
LIN {X 120.0436,Y -54.1037,Z 150,A -27.7769,B 24.249,C -1.2801,E1 24.426,E2 474.4962} C_DIS
LIN {X 118.4528,Y -57.5078,Z 150,A -29.3652,B 24.2491,C -1.2775,E1 24.4241,E2 476.0818} C_DIS
LIN {X 116.9645,Y -60.4774,Z 150,A -30.8025,B 24.2493,C -1.2736,E1 24.4223,E2 477.5208} C_DIS
LIN {X 115.4061,Y -63.4005,Z 150,A -32.2379,B 24.2495,C -1.2696,E1 24.4204,E2 478.9581} C_DIS
LIN {X 113.4056,Y -66.9124,Z 150,A -34.0799,B 24.25,C -1.26,E1 24.4178,E2 480.8135} C_DIS
LIN {X 111.1242,Y -70.6373,Z 150,A -35.8748,B 24.25,C -1.26,E1 24.4152,E2 482.5988} C_DIS
LIN {X 109.312,Y -73.4102,Z 150,A -37.3445,B 24.2503,C -1.2544,E1 24.4129,E2 484.0745} C_DIS
LIN {X 106.8993,Y -76.8811,Z 150,A -39.1435,B 24.2504,C -1.2514,E1 24.41,E2 485.8718} C_DIS
LIN {X 104.8848,Y -79.6074,Z 150,A -40.604,B 24.2506,C -1.2481,E1 24.4076,E2 487.3331} C_DIS
LIN {X 102.7971,Y -82.2856,Z 150,A -42.0802,B 24.2508,C -1.2442,E1 24.405,E2 488.8117} C_DIS
LIN {X 100.6539,Y -84.8937,Z 150,A -43.6057,B 24.2511,C -1.2373,E1 24.4023,E2 490.3467} C_DIS
LIN {X 97.8009,Y -88.1657,Z 150,A -45.4721,B 24.2513,C -1.2335,E1 24.3988,E2 492.2135} C_DIS
LIN {X 94.9399,Y -91.2391,Z 150,A -47.2538,B 24.2513,C -1.2313,E1 24.3954,E2 493.9926} C_DIS
LIN {X 92.034,Y -94.1691,Z 150,A -49.0579,B 24.2516,C -1.2264,E1 24.3918,E2 495.8006} C_DIS
LIN {X 88.9043,Y -97.1294,Z 150,A -50.9542,B 24.2519,C -1.2207,E1 24.3879,E2 497.7027} C_DIS
LIN {X 85.6073,Y -100.048,Z 150,A -52.7872,B 24.2519,C -1.2207,E1 24.3841,E2 499.5285} C_DIS
LIN {X 82.6832,Y -102.4769,Z 150,A -54.5035,B 24.2522,C -1.2137,E1 24.3804,E2 501.255} C_DIS
LIN {X 79.4089,Y -105.0346,Z 150,A -56.3134,B 24.2524,C -1.2096,E1 24.3763,E2 503.0678} C_DIS
LIN {X 75.9706,Y -107.5477,Z 150,A -58.1599,B 24.2526,C -1.2061,E1 24.3722,E2 504.9162} C_DIS
LIN {X 72.7581,Y -109.7473,Z 150,A -59.7555,B 24.2525,C -1.2078,E1 24.3685,E2 506.5021} C_DIS
LIN {X 69.9761,Y -111.5415,Z 150,A -61.3075,B 24.2529,C -1.1992,E1 24.3648,E2 508.0698} C_DIS
LIN {X 66.2809,Y -113.7761,Z 150,A -63.2038,B 24.2531,C -1.1948,E1 24.3602,E2 509.9708} C_DIS
LIN {X 62.6871,Y -115.7952,Z 150,A -64.9812,B 24.2532,C -1.1924,E1 24.3559,E2 511.7486} C_DIS
LIN {X 59.2113,Y -117.609,Z 150,A -66.5552,B 24.253,C -1.1963,E1 24.352,E2 513.3085} C_DIS
LIN {X 56.12,Y -119.1158,Z 150,A -68.0276,B 24.253,C -1.1951,E1 24.3483,E2 514.7799} C_DIS
LIN {X 53.5212,Y -120.3041,Z 150,A -69.2894,B 24.2532,C -1.1923,E1 24.3451,E2 516.0453} C_DIS
LIN {X 49.9865,Y -121.8177,Z 150,A -70.9426,B 24.2532,C -1.1908,E1 24.3408,E2 517.6982} C_DIS
LIN {X 47.0862,Y -122.967,Z 150,A -72.2791,B 24.2533,C -1.19,E1 24.3373,E2 519.0335} C_DIS
LIN {X 44.3463,Y -123.9801,Z 150,A -73.5646,B 24.2534,C -1.1876,E1 24.334,E2 520.3221} C_DIS
LIN {X 41.1692,Y -125.0714,Z 150,A -74.998,B 24.2534,C -1.1872,E1 24.3302,E2 521.7537} C_DIS
LIN {X 37.8758,Y -126.1089,Z 150,A -76.5012,B 24.2535,C -1.1853,E1 24.3262,E2 523.2586} C_DIS
LIN {X 35.1927,Y -126.8823,Z 150,A -77.7719,B 24.2537,C -1.1812,E1 24.3227,E2 524.5372} C_DIS
LIN {X 31.6236,Y -127.8208,Z 150,A -79.3235,B 24.2537,C -1.1822,E1 24.3185,E2 526.0837} C_DIS
LIN {X 28.774,Y -128.4911,Z 150,A -80.5451,B 24.2537,C -1.1837,E1 24.3152,E2 527.3001} C_DIS
LIN {X 26.1765,Y -129.0441,Z 150,A -81.7375,B 24.2537,C -1.1808,E1 24.312,E2 528.4979} C_DIS
LIN {X 22.988,Y -129.6503,Z 150,A -83.1528,B 24.2538,C -1.1795,E1 24.3081,E2 529.9147} C_DIS
LIN {X 19.7653,Y -130.181,Z 150,A -84.5903,B 24.2538,C -1.1776,E1 24.3041,E2 531.3554} C_DIS
LIN {X 16.3526,Y -130.6553,Z 150,A -86.0631,B 24.2538,C -1.1779,E1 24.3,E2 532.8261} C_DIS
LIN {X 13.4413,Y -130.9862,Z 150,A -87.4807,B 24.2542,C -1.17,E1 24.296,E2 534.262} C_DIS
LIN {X 9.6434,Y -131.3189,Z 150,A -89.0292,B 24.254,C -1.1748,E1 24.2918,E2 535.798} C_DIS
LIN {X 6.1655,Y -131.5289,Z 150,A -90.5125,B 24.254,C -1.1758,E1 24.2876,E2 537.2783} C_DIS
LIN {X 1.9359,Y -131.6586,Z 150,A -92.3736,B 24.254,C -1.1743,E1 24.2824,E2 539.1428} C_DIS
LIN {X 1.9359,Y -131.6586,Z 150,A -92.3736,B 24.254,C -1.1743,E1 24.2824,E2 539.1428} C_DIS
Enddeposition()
LIN {X 0.9326,Y -130.7208,Z 150,A -92.5095,B 23.2243,C -1.0032,E1 23.2452,E2 539.5748} C_DIS
Startdeposition()
$VEL.CP = VEL_PRINT
LIN {X 3.4072,Y -130.6814,Z 150,A -90.9979,B 23.2234,C -1.0238,E1 23.2496,E2 538.0111} C_DIS
LIN {X 6.3089,Y -130.5735,Z 150,A -89.4645,B 23.2229,C -1.0368,E1 23.2539,E2 536.4453} C_DIS
LIN {X 10.1232,Y -130.3344,Z 150,A -87.7105,B 23.2227,C -1.0414,E1 23.2588,E2 534.6807} C_DIS
LIN {X 14.9414,Y -129.8695,Z 150,A -85.316,B 23.2221,C -1.0559,E1 23.2656,E2 532.2512} C_DIS
LIN {X 18.4934,Y -129.4107,Z 150,A -84.0635,B 23.2227,C -1.0414,E1 23.2689,E2 531.0364} C_DIS
LIN {X 22.9197,Y -128.7005,Z 150,A -82.1664,B 23.2227,C -1.0396,E1 23.2741,E2 529.146} C_DIS
LIN {X 30.8606,Y -127.0306,Z 150,A -78.588,B 23.2226,C -1.0438,E1 23.2839,E2 525.5621} C_DIS
LIN {X 34.9363,Y -125.9707,Z 150,A -76.7618,B 23.2226,C -1.0448,E1 23.2888,E2 523.7366} C_DIS
LIN {X 38.1229,Y -125.043,Z 150,A -75.2571,B 23.2223,C -1.0489,E1 23.2929,E2 522.2243} C_DIS
LIN {X 42.3386,Y -123.6801,Z 150,A -73.3414,B 23.2223,C -1.05,E1 23.298,E2 520.3099} C_DIS
LIN {X 45.5556,Y -122.531,Z 150,A -72.1007,B 23.2228,C -1.0394,E1 23.3011,E2 519.0988} C_DIS
LIN {X 47.4798,Y -121.798,Z 150,A -70.3447,B 23.2209,C -1.0829,E1 23.306,E2 517.237} C_DIS
LIN {X 52.1439,Y -119.8755,Z 150,A -68.9404,B 23.2225,C -1.0461,E1 23.3093,E2 515.9296} C_DIS
LIN {X 56.031,Y -118.1088,Z 150,A -66.9741,B 23.2221,C -1.0537,E1 23.3144,E2 513.9494} C_DIS
LIN {X 59.0607,Y -116.623,Z 150,A -65.4346,B 23.2219,C -1.0591,E1 23.3182,E2 512.4007} C_DIS
LIN {X 61.9936,Y -115.0928,Z 150,A -63.0203,B 23.2197,C -1.1099,E1 23.3245,E2 509.8653} C_DIS
LIN {X 67.8781,Y -111.7237,Z 150,A -60.9482,B 23.2214,C -1.0701,E1 23.3292,E2 507.901} C_DIS
LIN {X 72.6107,Y -108.7071,Z 150,A -58.5558,B 23.2214,C -1.0715,E1 23.3348,E2 505.5134} C_DIS
LIN {X 75.7396,Y -106.5513,Z 150,A -56.8049,B 23.221,C -1.0792,E1 23.3388,E2 503.7497} C_DIS
LIN {X 79.4742,Y -103.795,Z 150,A -54.8754,B 23.221,C -1.0783,E1 23.3431,E2 501.8302} C_DIS
LIN {X 81.7403,Y -102.0208,Z 150,A -53.5814,B 23.2209,C -1.0826,E1 23.3459,E2 500.5304} C_DIS
LIN {X 85.073,Y -99.2583,Z 150,A -51.7173,B 23.2208,C -1.0853,E1 23.3499,E2 498.6675} C_DIS
LIN {X 88.1713,Y -96.5169,Z 150,A -49.8606,B 23.2205,C -1.0917,E1 23.3538,E2 496.8027} C_DIS
LIN {X 91.2887,Y -93.5737,Z 150,A -48.2732,B 23.2209,C -1.0815,E1 23.3569,E2 495.2481} C_DIS
LIN {X 93.3092,Y -91.5584,Z 150,A -46.6314,B 23.2199,C -1.1043,E1 23.3602,E2 493.5563} C_DIS
LIN {X 96.7436,Y -87.9217,Z 150,A -44.5904,B 23.22,C -1.1022,E1 23.3641,E2 491.5304} C_DIS
LIN {X 99.6693,Y -84.5907,Z 150,A -42.9538,B 23.2205,C -1.0917,E1 23.367,E2 489.9282} C_DIS
LIN {X 102.4238,Y -81.234,Z 150,A -40.7711,B 23.2196,C -1.1109,E1 23.3709,E2 487.7081} C_DIS
LIN {X 104.8037,Y -78.1391,Z 150,A -38.747,B 23.2187,C -1.1315,E1 23.3744,E2 485.6425} C_DIS
LIN {X 107.0388,Y -75.0492,Z 150,A -37.4867,B 23.2194,C -1.1152,E1 23.3763,E2 484.4302} C_DIS
LIN {X 109.2748,Y -71.7537,Z 150,A -35.7406,B 23.2192,C -1.1201,E1 23.379,E2 482.681} C_DIS
LIN {X 111.3817,Y -68.4374,Z 150,A -33.9903,B 23.2189,C -1.1265,E1 23.3816,E2 480.9242} C_DIS
LIN {X 113.5104,Y -64.8455,Z 150,A -32.1473,B 23.2186,C -1.1325,E1 23.3842,E2 479.0764} C_DIS
LIN {X 115.3134,Y -61.583,Z 150,A -30.6034,B 23.2186,C -1.1327,E1 23.3863,E2 477.5407} C_DIS
LIN {X 116.7564,Y -58.7989,Z 150,A -29.2928,B 23.2186,C -1.1336,E1 23.3879,E2 476.2354} C_DIS
LIN {X 118.9629,Y -54.1978,Z 150,A -26.8844,B 23.2179,C -1.1491,E1 23.3908,E2 473.802} C_DIS
LIN {X 120.5008,Y -50.6825,Z 150,A -24.9047,B 23.2169,C -1.1696,E1 23.393,E2 471.7824} C_DIS
LIN {X 121.9933,Y -46.9773,Z 150,A -23.5185,B 23.2175,C -1.1563,E1 23.3944,E2 470.438} C_DIS
LIN {X 123.3978,Y -43.1528,Z 150,A -21.8083,B 23.2175,C -1.158,E1 23.396,E2 468.7339} C_DIS
LIN {X 124.4827,Y -39.9144,Z 150,A -20.5502,B 23.2178,C -1.1505,E1 23.3971,E2 467.5024} C_DIS
LIN {X 126.3964,Y -33.3639,Z 150,A -17.2822,B 23.2167,C -1.1741,E1 23.3996,E2 464.1952} C_DIS
LIN {X 127.4185,Y -29.2172,Z 150,A -15.4258,B 23.2164,C -1.1793,E1 23.4008,E2 462.3374} C_DIS
LIN {X 128.2782,Y -25.1838,Z 150,A -13.5901,B 23.2161,C -1.1866,E1 23.4018,E2 460.4951} C_DIS
LIN {X 128.9755,Y -21.3187,Z 150,A -11.9606,B 23.2161,C -1.1874,E1 23.4026,E2 458.8737} C_DIS
LIN {X 129.5792,Y -17.2756,Z 150,A -10.23,B 23.2159,C -1.1901,E1 23.4033,E2 457.1475} C_DIS
LIN {X 130.1156,Y -12.6135,Z 150,A -8.1624,B 23.2156,C -1.1974,E1 23.4039,E2 455.0749} C_DIS
LIN {X 130.379,Y -9.512,Z 150,A -6.8026,B 23.2154,C -1.2016,E1 23.4042,E2 453.7132} C_DIS
LIN {X 130.6178,Y -5.3107,Z 150,A -4.9887,B 23.2151,C -1.206,E1 23.4044,E2 451.8998} C_DIS
LIN {X 130.7198,Y -1.4194,Z 150,A -3.276,B 23.2149,C -1.2119,E1 23.4045,E2 450.1834} C_DIS
LIN {X 130.6997,Y 2.6422,Z 150,A -1.4071,B 23.2143,C -1.2222,E1 23.4045,E2 448.3006} C_DIS
LIN {X 130.5508,Y 6.761,Z 150,A 0.3267,B 23.2143,C -1.2243,E1 23.4042,E2 446.5726} C_DIS
LIN {X 130.2667,Y 10.9429,Z 150,A 1.9443,B 23.2145,C -1.219,E1 23.4039,E2 444.9786} C_DIS
LIN {X 129.9756,Y 13.9819,Z 150,A 3.6136,B 23.2134,C -1.2402,E1 23.4034,E2 443.2666} C_DIS
LIN {X 129.3906,Y 18.6339,Z 150,A 5.4723,B 23.2136,C -1.2368,E1 23.4027,E2 441.4287} C_DIS
LIN {X 128.7128,Y 22.851,Z 150,A 7.8254,B 23.2121,C -1.2673,E1 23.4016,E2 439.0135} C_DIS
LIN {X 127.8605,Y 27.22,Z 150,A 9.2935,B 23.213,C -1.2487,E1 23.4008,E2 437.6016} C_DIS
LIN {X 126.943,Y 31.2242,Z 150,A 11.138,B 23.2126,C -1.2565,E1 23.3995,E2 435.7489} C_DIS
LIN {X 125.9696,Y 34.9402,Z 150,A 12.7082,B 23.2126,C -1.256,E1 23.3984,E2 434.1899} C_DIS
LIN {X 125.0169,Y 38.2082,Z 150,A 14.1837,B 23.2124,C -1.2597,E1 23.3972,E2 432.7142} C_DIS
LIN {X 123.9757,Y 41.4622,Z 150,A 15.6854,B 23.2122,C -1.2644,E1 23.3959,E2 431.2098} C_DIS
LIN {X 122.5503,Y 45.5042,Z 150,A 17.5288,B 23.212,C -1.2683,E1 23.3942,E2 429.3679} C_DIS
LIN {X 121.6372,Y 47.8932,Z 150,A 19.2122,B 23.2103,C -1.3001,E1 23.3924,E2 427.6142} C_DIS
LIN {X 119.8831,Y 52.1264,Z 150,A 20.6628,B 23.2115,C -1.2776,E1 23.3909,E2 426.229} C_DIS
LIN {X 117.3715,Y 57.5591,Z 150,A 23.2913,B 23.2111,C -1.2853,E1 23.3877,E2 423.5964} C_DIS
LIN {X 115.8357,Y 60.5902,Z 150,A 24.7217,B 23.2111,C -1.2865,E1 23.3859,E2 422.1712} C_DIS
LIN {X 113.8246,Y 64.293,Z 150,A 26.7237,B 23.2104,C -1.2994,E1 23.3831,E2 420.1481} C_DIS
LIN {X 111.3727,Y 68.452,Z 150,A 28.7491,B 23.2104,C -1.3005,E1 23.3802,E2 418.1311} C_DIS
LIN {X 108.931,Y 72.2752,Z 150,A 30.8614,B 23.2097,C -1.3119,E1 23.377,E2 416.0015} C_DIS
LIN {X 106.0962,Y 76.3761,Z 150,A 32.9296,B 23.2097,C -1.3116,E1 23.3737,E2 413.9451} C_DIS
LIN {X 103.5578,Y 79.7839,Z 150,A 34.7528,B 23.2096,C -1.3143,E1 23.3706,E2 412.1246} C_DIS
LIN {X 101.009,Y 82.987,Z 150,A 36.5776,B 23.2093,C -1.3201,E1 23.3674,E2 410.2943} C_DIS
LIN {X 98.1154,Y 86.3886,Z 150,A 38.3903,B 23.2094,C -1.3174,E1 23.3641,E2 408.4972} C_DIS
LIN {X 95.2333,Y 89.5556,Z 150,A 40.358,B 23.2089,C -1.3262,E1 23.3603,E2 406.5167} C_DIS
LIN {X 92.1921,Y 92.6831,Z 150,A 41.9858,B 23.2095,C -1.3163,E1 23.3572,E2 404.9216} C_DIS
LIN {X 90.2721,Y 94.5541,Z 150,A 43.2706,B 23.2091,C -1.3242,E1 23.3546,E2 403.6225} C_DIS
LIN {X 87.0744,Y 97.507,Z 150,A 45.3262,B 23.2084,C -1.3354,E1 23.3503,E2 401.5476} C_DIS
LIN {X 83.6885,Y 100.4288,Z 150,A 47.3113,B 23.2082,C -1.3405,E1 23.3461,E2 399.5581} C_DIS
LIN {X 80.2307,Y 103.2115,Z 150,A 49.2198,B 23.2081,C -1.3423,E1 23.3419,E2 397.6527} C_DIS
LIN {X 76.6843,Y 105.8729,Z 150,A 51.1171,B 23.2081,C -1.3435,E1 23.3377,E2 395.7597} C_DIS
LIN {X 72.19,Y 108.9875,Z 150,A 53.5808,B 23.2076,C -1.3508,E1 23.332,E2 393.2867} C_DIS
LIN {X 69.3258,Y 110.8312,Z 150,A 55.2101,B 23.2071,C -1.3598,E1 23.3281,E2 391.6401} C_DIS
LIN {X 64.8712,Y 113.4957,Z 150,A 57.2737,B 23.2075,C -1.3528,E1 23.3231,E2 389.6011} C_DIS
LIN {X 60.9281,Y 115.6582,Z 150,A 59.8291,B 23.2058,C -1.3841,E1 23.3167,E2 386.9742} C_DIS
LIN {X 56.3722,Y 117.9458,Z 150,A 61.4905,B 23.2072,C -1.3589,E1 23.3127,E2 385.3814} C_DIS
LIN {X 52.3468,Y 119.7878,Z 150,A 63.1964,B 23.2077,C -1.3498,E1 23.3084,E2 383.7032} C_DIS
LIN {X 49.1917,Y 121.1171,Z 150,A 64.6282,B 23.2077,C -1.3481,E1 23.3047,E2 382.2794} C_DIS
LIN {X 45.9155,Y 122.3962,Z 150,A 66.3213,B 23.2073,C -1.3569,E1 23.3003,E2 380.5679} C_DIS
LIN {X 42.9812,Y 123.4573,Z 150,A 67.7191,B 23.2071,C -1.3596,E1 23.2966,E2 379.1664} C_DIS
LIN {X 39.8829,Y 124.4927,Z 150,A 69.1516,B 23.2071,C -1.3609,E1 23.2928,E2 377.7337} C_DIS
LIN {X 36.7797,Y 125.4446,Z 150,A 70.5804,B 23.207,C -1.3622,E1 23.2889,E2 376.3041} C_DIS
LIN {X 33.6035,Y 126.3325,Z 150,A 71.9325,B 23.2072,C -1.3588,E1 23.2853,E2 374.9633} C_DIS
LIN {X 30.5639,Y 127.1021,Z 150,A 73.1756,B 23.2075,C -1.3533,E1 23.282,E2 373.7359} C_DIS
LIN {X 24.6881,Y 128.373,Z 150,A 75.7503,B 23.2075,C -1.3517,E1 23.275,E2 371.1688} C_DIS
LIN {X 20.9683,Y 129.034,Z 150,A 77.6902,B 23.2068,C -1.3658,E1 23.2696,E2 369.1955} C_DIS
LIN {X 17.4381,Y 129.5579,Z 150,A 79.3278,B 23.2066,C -1.3697,E1 23.265,E2 367.5495} C_DIS
LIN {X 13.5486,Y 130.0222,Z 150,A 81.049,B 23.2066,C -1.3702,E1 23.2602,E2 365.8284} C_DIS
LIN {X 8.5678,Y 130.4455,Z 150,A 83.3166,B 23.2063,C -1.374,E1 23.2539,E2 363.5525} C_DIS
LIN {X 4.3043,Y 130.6564,Z 150,A 85.1336,B 23.2065,C -1.3713,E1 23.2489,E2 361.7427} C_DIS
LIN {X 0.5182,Y 130.7248,Z 150,A 86.7085,B 23.2067,C -1.3671,E1 23.2445,E2 360.1787} C_DIS
LIN {X -4.6677,Y 130.6429,Z 150,A 89.0116,B 23.2067,C -1.3679,E1 23.238,E2 357.8733} C_DIS
LIN {X -10.3246,Y 130.3189,Z 150,A 91.5585,B 23.2066,C -1.3699,E1 23.2309,E2 355.3204} C_DIS
LIN {X -14.0538,Y 129.9678,Z 150,A 93.0301,B 23.207,C -1.3612,E1 23.2269,E2 353.8701} C_DIS
LIN {X -17.2717,Y 129.5797,Z 150,A 94.5119,B 23.207,C -1.3632,E1 23.2228,E2 352.382} C_DIS
LIN {X -21.2955,Y 128.9794,Z 150,A 96.8422,B 23.2056,C -1.3874,E1 23.2162,E2 349.9878} C_DIS
LIN {X -25.7256,Y 128.1695,Z 150,A 98.3215,B 23.2069,C -1.3629,E1 23.2123,E2 348.5692} C_DIS
LIN {X -29.9437,Y 127.2516,Z 150,A 100.3103,B 23.2068,C -1.3656,E1 23.2069,E2 346.5706} C_DIS
LIN {X -34.4472,Y 126.1075,Z 150,A 102.3429,B 23.2069,C -1.3634,E1 23.2014,E2 344.5403} C_DIS
LIN {X -38.1441,Y 125.0365,Z 150,A 103.7848,B 23.2076,C -1.3503,E1 23.1976,E2 343.129} C_DIS
LIN {X -47.7057,Y 121.7101,Z 150,A 108.2749,B 23.2078,C -1.347,E1 23.1858,E2 338.6378} C_DIS
LIN {X -53.8486,Y 119.1203,Z 150,A 111.4262,B 23.2075,C -1.3532,E1 23.1776,E2 335.4628} C_DIS
LIN {X -57.6423,Y 117.3305,Z 150,A 113.0992,B 23.208,C -1.3428,E1 23.1735,E2 333.8116} C_DIS
LIN {X -60.4198,Y 115.9251,Z 150,A 114.3219,B 23.2085,C -1.3342,E1 23.1705,E2 332.6072} C_DIS
LIN {X -63.8579,Y 114.0691,Z 150,A 116.3119,B 23.208,C -1.3437,E1 23.1655,E2 330.5867} C_DIS
LIN {X -67.5691,Y 111.9105,Z 150,A 118.333,B 23.2078,C -1.3466,E1 23.1606,E2 328.5515} C_DIS
LIN {X -71.7875,Y 109.2525,Z 150,A 120.4049,B 23.2083,C -1.3373,E1 23.1558,E2 326.496} C_DIS
LIN {X -77.2155,Y 105.4863,Z 150,A 123.7687,B 23.2075,C -1.3526,E1 23.1481,E2 323.0807} C_DIS
LIN {X -80.82,Y 102.7505,Z 150,A 125.2886,B 23.2089,C -1.3275,E1 23.1448,E2 321.6188} C_DIS
LIN {X -86.7706,Y 97.7776,Z 150,A 129.466,B 23.2074,C -1.3549,E1 23.1358,E2 317.3537} C_DIS
LIN {X -91.1689,Y 93.6903,Z 150,A 131.1926,B 23.2099,C -1.308,E1 23.1326,E2 315.739} C_DIS
LIN {X -96.4688,Y 88.2237,Z 150,A 134.6888,B 23.2099,C -1.3068,E1 23.1258,E2 312.2295} C_DIS
LIN {X -99.1607,Y 85.1864,Z 150,A 136.4968,B 23.2102,C -1.3035,E1 23.1225,E2 310.4209} C_DIS
LIN {X -102.0025,Y 81.763,Z 150,A 138.4087,B 23.2105,C -1.2967,E1 23.1191,E2 308.5168} C_DIS
LIN {X -104.5768,Y 78.4435,Z 150,A 140.3067,B 23.2107,C -1.2943,E1 23.1159,E2 306.6151} C_DIS
LIN {X -107.2445,Y 74.754,Z 150,A 142.3235,B 23.2109,C -1.2897,E1 23.1126,E2 304.5992} C_DIS
LIN {X -110.5082,Y 69.839,Z 150,A 144.8672,B 23.2114,C -1.2806,E1 23.1088,E2 302.0649} C_DIS
LIN {X -112.6556,Y 66.3194,Z 150,A 146.7615,B 23.2114,C -1.2792,E1 23.106,E2 300.1634} C_DIS
LIN {X -114.9421,Y 62.2735,Z 150,A 148.7845,B 23.2118,C -1.2727,E1 23.1033,E2 298.1457} C_DIS
LIN {X -116.276,Y 59.7424,Z 150,A 149.8269,B 23.2124,C -1.2597,E1 23.102,E2 297.1303} C_DIS
LIN {X -117.4951,Y 57.3086,Z 150,A 151.0504,B 23.2126,C -1.2574,E1 23.1005,E2 295.9054} C_DIS
LIN {X -119.1603,Y 53.759,Z 150,A 152.941,B 23.2124,C -1.2598,E1 23.0983,E2 293.9975} C_DIS
LIN {X -120.5586,Y 50.5441,Z 150,A 154.4655,B 23.2127,C -1.2546,E1 23.0966,E2 292.4771} C_DIS
LIN {X -122.1273,Y 46.6321,Z 150,A 156.379,B 23.2129,C -1.2518,E1 23.0946,E2 290.5592} C_DIS
LIN {X -123.4022,Y 43.1402,Z 150,A 157.993,B 23.2131,C -1.2461,E1 23.0931,E2 288.9499} C_DIS
LIN {X -124.5159,Y 39.8103,Z 150,A 159.4685,B 23.2135,C -1.2385,E1 23.0918,E2 287.4845} C_DIS
LIN {X -125.6195,Y 36.1823,Z 150,A 161.3892,B 23.2132,C -1.2446,E1 23.0903,E2 285.5363} C_DIS
LIN {X -126.8653,Y 31.539,Z 150,A 163.3875,B 23.2138,C -1.2331,E1 23.0889,E2 283.5547} C_DIS
LIN {X -127.7164,Y 27.8876,Z 150,A 164.9977,B 23.2141,C -1.2264,E1 23.088,E2 281.9513} C_DIS
LIN {X -128.4107,Y 24.4909,Z 150,A 166.4644,B 23.2145,C -1.2192,E1 23.0872,E2 280.4935} C_DIS
LIN {X -129.0764,Y 20.7104,Z 150,A 168.2733,B 23.2145,C -1.2192,E1 23.0863,E2 278.6728} C_DIS
LIN {X -129.5988,Y 17.126,Z 150,A 170.196,B 23.214,C -1.2289,E1 23.0856,E2 276.7129} C_DIS
LIN {X -130.0519,Y 13.2629,Z 150,A 171.4554,B 23.2153,C -1.2038,E1 23.0852,E2 275.5095} C_DIS
LIN {X -130.6056,Y 5.6253,Z 150,A 174.7496,B 23.2159,C -1.1901,E1 23.0846,E2 272.2288} C_DIS
LIN {X -130.7224,Y -1.015,Z 150,A 177.5825,B 23.2165,C -1.1772,E1 23.0846,E2 269.4103} C_DIS
LIN {X -130.5357,Y -7.0601,Z 150,A -179.5532,B 23.2165,C -1.1779,E1 23.0848,E2 266.5254} C_DIS
LIN {X -130.362,Y -9.7449,Z 150,A -177.4052,B 23.2146,C -1.217,E1 23.0853,E2 264.2634} C_DIS
LIN {X -129.721,Y -16.1899,Z 150,A -175.336,B 23.2167,C -1.1737,E1 23.086,E2 262.2914} C_DIS
LIN {X -129.1722,Y -20.092,Z 150,A -173.7083,B 23.2172,C -1.1639,E1 23.0866,E2 260.6783} C_DIS
LIN {X -128.4536,Y -24.2665,Z 150,A -171.8178,B 23.2174,C -1.1595,E1 23.0875,E2 258.7868} C_DIS
LIN {X -127.7668,Y -27.654,Z 150,A -170.3341,B 23.2177,C -1.1534,E1 23.0884,E2 257.3091} C_DIS
LIN {X -126.8767,Y -31.494,Z 150,A -168.5325,B 23.2177,C -1.1513,E1 23.0896,E2 255.5015} C_DIS
LIN {X -126.0088,Y -34.8001,Z 150,A -167.0414,B 23.218,C -1.1464,E1 23.0907,E2 254.0134} C_DIS
LIN {X -125.0144,Y -38.2161,Z 150,A -165.5755,B 23.2184,C -1.1375,E1 23.0918,E2 252.561} C_DIS
LIN {X -124.0481,Y -41.2449,Z 150,A -163.918,B 23.2181,C -1.145,E1 23.0933,E2 250.8741} C_DIS
LIN {X -122.5476,Y -45.5113,Z 150,A -162.0537,B 23.2186,C -1.1339,E1 23.095,E2 249.0268} C_DIS
LIN {X -120.8956,Y -49.7372,Z 150,A -159.997,B 23.2187,C -1.131,E1 23.0972,E2 246.9648} C_DIS
LIN {X -119.3624,Y -53.3073,Z 150,A -158.3291,B 23.219,C -1.1246,E1 23.099,E2 245.3033} C_DIS
LIN {X -117.4713,Y -57.3569,Z 150,A -156.3778,B 23.2193,C -1.1187,E1 23.1014,E2 243.3557} C_DIS
LIN {X -115.4587,Y -61.308,Z 150,A -153.5172,B 23.2176,C -1.1546,E1 23.1053,E2 240.387} C_DIS
LIN {X -112.2165,Y -67.0598,Z 150,A -151.4892,B 23.2198,C -1.1077,E1 23.108,E2 238.4673} C_DIS
LIN {X -109.9289,Y -70.7479,Z 150,A -149.5672,B 23.22,C -1.1035,E1 23.1109,E2 236.5451} C_DIS
LIN {X -107.5697,Y -74.2862,Z 150,A -147.6653,B 23.22,C -1.1005,E1 23.1138,E2 234.6408} C_DIS
LIN {X -105.059,Y -77.7964,Z 150,A -145.7594,B 23.2203,C -1.0964,E1 23.117,E2 232.7352} C_DIS
LIN {X -102.3611,Y -81.3128,Z 150,A -143.8228,B 23.2205,C -1.0914,E1 23.1203,E2 230.8014} C_DIS
LIN {X -99.5073,Y -84.7812,Z 150,A -141.948,B 23.2209,C -1.0826,E1 23.1236,E2 228.9398} C_DIS
LIN {X -94.7884,Y -90.0269,Z 150,A -138.8122,B 23.2211,C -1.0775,E1 23.1296,E2 225.8019} C_DIS
LIN {X -91.6571,Y -93.2123,Z 150,A -136.7823,B 23.2211,C -1.0766,E1 23.1336,E2 223.7649} C_DIS
LIN {X -88.5681,Y -96.1522,Z 150,A -134.8824,B 23.2213,C -1.0741,E1 23.1374,E2 221.8629} C_DIS
LIN {X -85.1408,Y -99.2,Z 150,A -132.8943,B 23.2215,C -1.0691,E1 23.1416,E2 219.879} C_DIS
LIN {X -81.9124,Y -101.882,Z 150,A -131.0251,B 23.2215,C -1.067,E1 23.1457,E2 218.0074} C_DIS
LIN {X -78.1111,Y -104.8246,Z 150,A -128.1052,B 23.2201,C -1.1009,E1 23.1524,E2 214.99} C_DIS
LIN {X -72.9652,Y -108.4701,Z 150,A -125.9585,B 23.2215,C -1.0676,E1 23.1572,E2 212.9203} C_DIS
LIN {X -68.6283,Y -111.2645,Z 150,A -123.8329,B 23.222,C -1.0578,E1 23.1622,E2 210.8122} C_DIS
LIN {X -64.7073,Y -113.5893,Z 150,A -121.8761,B 23.2222,C -1.053,E1 23.1669,E2 208.8612} C_DIS
LIN {X -61.5296,Y -115.3421,Z 150,A -120.1967,B 23.2221,C -1.055,E1 23.171,E2 207.1717} C_DIS
LIN {X -57.3525,Y -117.4735,Z 150,A -118.3146,B 23.2225,C -1.0444,E1 23.1757,E2 205.3111} C_DIS
LIN {X -54.2297,Y -118.9482,Z 150,A -116.6529,B 23.2223,C -1.0495,E1 23.1799,E2 203.6319} C_DIS
LIN {X -51.1112,Y -120.3218,Z 150,A -115.1003,B 23.2223,C -1.0506,E1 23.1839,E2 202.0725} C_DIS
LIN {X -47.3837,Y -121.8353,Z 150,A -113.5329,B 23.2227,C -1.0398,E1 23.1879,E2 200.5291} C_DIS
LIN {X -44.3451,Y -122.9739,Z 150,A -112.0989,B 23.2227,C -1.039,E1 23.1917,E2 199.0938} C_DIS
LIN {X -41.0833,Y -124.1019,Z 150,A -110.5424,B 23.2227,C -1.0398,E1 23.1958,E2 197.5322} C_DIS
LIN {X -37.0185,Y -125.3746,Z 150,A -108.7637,B 23.223,C -1.0343,E1 23.2006,E2 195.7642} C_DIS
LIN {X -33.9415,Y -126.2424,Z 150,A -107.3217,B 23.223,C -1.0353,E1 23.2045,E2 194.3172} C_DIS
LIN {X -29.2024,Y -127.4219,Z 150,A -105.1567,B 23.223,C -1.0353,E1 23.2103,E2 192.1491} C_DIS
LIN {X -23.82,Y -128.5389,Z 150,A -102.7829,B 23.223,C -1.0325,E1 23.2168,E2 189.7793} C_DIS
LIN {X -20.1367,Y -129.1652,Z 150,A -101.099,B 23.223,C -1.0342,E1 23.2215,E2 188.0893} C_DIS
LIN {X -16.5776,Y -129.6707,Z 150,A -99.4199,B 23.2228,C -1.0388,E1 23.2262,E2 186.3972} C_DIS
LIN {X -12.0777,Y -130.167,Z 150,A -97.4272,B 23.2228,C -1.039,E1 23.2317,E2 184.4028} C_DIS
LIN {X -7.3074,Y -130.5232,Z 150,A -95.3238,B 23.2228,C -1.0393,E1 23.2376,E2 182.2979} C_DIS
LIN {X -3.2324,Y -130.6862,Z 150,A -93.5579,B 23.2228,C -1.0385,E1 23.2425,E2 180.5338} C_DIS
LIN {X 0.9326,Y -130.7208,Z 150,A -92.5061,B 23.2243,C -1.0019,E1 23.2452,E2 179.5748} C_DIS
Enddeposition()
LIN {X 0.9326,Y -130.7208,Z 150,A -92.5061,B 23.2243,C -1.0019,E1 23.2452,E2 179.5748} C_DIS
Startdeposition()
$VEL.CP = VEL_PRINT
LIN {X -1.479,Y -129.772,Z 150,A -93.3957,B 22.3098,C -0.8579,E1 22.3226,E2 180.7276} C_DIS
LIN {X -5.291,Y -129.6709,Z 150,A -95.0778,B 22.3098,C -0.8579,E1 22.3179,E2 182.4103} C_DIS
LIN {X -10.6964,Y -129.3372,Z 150,A -97.7393,B 22.3102,C -0.8458,E1 22.3104,E2 185.1046} C_DIS
LIN {X -14.2551,Y -128.9937,Z 150,A -98.7088,B 22.3092,C -0.8732,E1 22.308,E2 186.0025} C_DIS
LIN {X -16.7817,Y -128.6889,Z 150,A -100.0744,B 22.3096,C -0.8626,E1 22.3041,E2 187.3973} C_DIS
LIN {X -20.4757,Y -128.1545,Z 150,A -101.6911,B 22.3096,C -0.8644,E1 22.2996,E2 189.0107} C_DIS
LIN {X -24.4732,Y -127.45,Z 150,A -103.5937,B 22.3096,C -0.8602,E1 22.2944,E2 190.9267} C_DIS
LIN {X -29.1973,Y -126.4516,Z 150,A -105.9121,B 22.31,C -0.853,E1 22.288,E2 193.2675} C_DIS
LIN {X -33.8467,Y -125.2876,Z 150,A -107.8816,B 22.3097,C -0.8607,E1 22.2827,E2 195.2198} C_DIS
LIN {X -37.7923,Y -124.1538,Z 150,A -109.5964,B 22.3095,C -0.8663,E1 22.2781,E2 196.9231} C_DIS
LIN {X -40.9023,Y -123.1641,Z 150,A -111.0677,B 22.3095,C -0.8661,E1 22.2742,E2 198.398} C_DIS
LIN {X -44.1643,Y -122.0324,Z 150,A -112.5285,B 22.3093,C -0.8702,E1 22.2704,E2 199.8511} C_DIS
LIN {X -47.1238,Y -120.9203,Z 150,A -113.9381,B 22.3093,C -0.871,E1 22.2667,E2 201.2621} C_DIS
LIN {X -50.9045,Y -119.3797,Z 150,A -115.7565,B 22.3093,C -0.8721,E1 22.262,E2 203.0822} C_DIS
LIN {X -54.7502,Y -117.6642,Z 150,A -117.5409,B 22.3091,C -0.8775,E1 22.2575,E2 204.8573} C_DIS
LIN {X -57.333,Y -116.4271,Z 150,A -118.889,B 22.3091,C -0.8754,E1 22.2541,E2 206.2149} C_DIS
LIN {X -60.8311,Y -114.6396,Z 150,A -120.5952,B 22.3091,C -0.8788,E1 22.2499,E2 207.9173} C_DIS
LIN {X -64.0503,Y -112.8738,Z 150,A -122.3788,B 22.3091,C -0.874,E1 22.2455,E2 209.7195} C_DIS
LIN {X -67.8854,Y -110.6093,Z 150,A -124.3192,B 22.3091,C -0.878,E1 22.2409,E2 211.656} C_DIS
LIN {X -70.6977,Y -108.8333,Z 150,A -125.602,B 22.3087,C -0.8883,E1 22.2379,E2 212.9163} C_DIS
LIN {X -73.6624,Y -106.8493,Z 150,A -127.5549,B 22.3092,C -0.8747,E1 22.2333,E2 214.9128} C_DIS
LIN {X -77.9234,Y -103.7829,Z 150,A -129.5574,B 22.3085,C -0.8922,E1 22.2289,E2 216.877} C_DIS
LIN {X -80.7018,Y -101.637,Z 150,A -131.269,B 22.3087,C -0.8881,E1 22.2251,E2 218.6065} C_DIS
LIN {X -84.1883,Y -98.7684,Z 150,A -133.2664,B 22.3085,C -0.8917,E1 22.2208,E2 220.603} C_DIS
LIN {X -87.5275,Y -95.8225,Z 150,A -135.2875,B 22.3085,C -0.8932,E1 22.2166,E2 222.6292} C_DIS
LIN {X -90.7414,Y -92.784,Z 150,A -137.221,B 22.3083,C -0.8981,E1 22.2127,E2 224.5589} C_DIS
LIN {X -93.8976,Y -89.5885,Z 150,A -139.3989,B 22.3084,C -0.8942,E1 22.2084,E2 226.7579} C_DIS
LIN {X -97.5396,Y -85.6096,Z 150,A -141.6258,B 22.308,C -0.906,E1 22.2043,E2 228.9647} C_DIS
LIN {X -100.3114,Y -82.344,Z 150,A -143.5272,B 22.3078,C -0.91,E1 22.2009,E2 230.8654} C_DIS
LIN {X -103.1373,Y -78.7753,Z 150,A -145.5174,B 22.3076,C -0.9157,E1 22.1975,E2 232.8514} C_DIS
LIN {X -105.7899,Y -75.1764,Z 150,A -147.5332,B 22.3075,C -0.9188,E1 22.1942,E2 234.87} C_DIS
LIN {X -108.2851,Y -71.5347,Z 150,A -149.4953,B 22.3073,C -0.9233,E1 22.1911,E2 236.8315} C_DIS
LIN {X -110.776,Y -67.6136,Z 150,A -151.4975,B 22.307,C -0.9307,E1 22.1882,E2 238.8256} C_DIS
LIN {X -113.5757,Y -62.7966,Z 150,A -154.1704,B 22.3071,C -0.9284,E1 22.1845,E2 241.5204} C_DIS
LIN {X -115.7221,Y -58.7431,Z 150,A -155.939,B 22.3065,C -0.9447,E1 22.1822,E2 243.2566} C_DIS
LIN {X -117.2223,Y -55.6899,Z 150,A -157.4777,B 22.3063,C -0.9473,E1 22.1804,E2 244.7976} C_DIS
LIN {X -118.6602,Y -52.5579,Z 150,A -158.9746,B 22.3061,C -0.9527,E1 22.1786,E2 246.2897} C_DIS
LIN {X -120.19,Y -48.9587,Z 150,A -161.0696,B 22.3065,C -0.9424,E1 22.1764,E2 248.4252} C_DIS
LIN {X -121.42,Y -45.8219,Z 150,A -162.0181,B 22.3055,C -0.9691,E1 22.1755,E2 249.3091} C_DIS
LIN {X -123.257,Y -40.6233,Z 150,A -164.1828,B 22.3047,C -0.9875,E1 22.1735,E2 251.4389} C_DIS
LIN {X -124.0174,Y -38.2381,Z 150,A -165.7936,B 22.3054,C -0.9698,E1 22.1721,E2 253.1073} C_DIS
LIN {X -124.9559,Y -35.049,Z 150,A -167.2662,B 22.3053,C -0.974,E1 22.1709,E2 254.5783} C_DIS
LIN {X -125.8383,Y -31.736,Z 150,A -168.7668,B 22.305,C -0.9792,E1 22.1699,E2 256.0751} C_DIS
LIN {X -126.6028,Y -28.5355,Z 150,A -170.343,B 22.305,C -0.9785,E1 22.1689,E2 257.6635} C_DIS
LIN {X -127.4767,Y -24.3336,Z 150,A -172.2095,B 22.3048,C -0.9856,E1 22.1679,E2 259.5238} C_DIS
LIN {X -128.1966,Y -20.2035,Z 150,A -174.0774,B 22.3046,C -0.9907,E1 22.167,E2 261.3908} C_DIS
LIN {X -128.7506,Y -16.311,Z 150,A -175.9897,B 22.3046,C -0.9889,E1 22.1663,E2 263.3208} C_DIS
LIN {X -129.3653,Y -10.3629,Z 150,A -178.4985,B 22.3041,C -1.0027,E1 22.1656,E2 265.8102} C_DIS
LIN {X -129.6102,Y -6.609,Z 150,A 179.8728,B 22.3038,C -1.0093,E1 22.1654,E2 267.4325} C_DIS
LIN {X -129.7623,Y -2.0581,Z 150,A 177.8297,B 22.3035,C -1.0144,E1 22.1652,E2 269.476} C_DIS
LIN {X -129.7101,Y 4.2686,Z 150,A 175.1303,B 22.303,C -1.0272,E1 22.1653,E2 272.1599} C_DIS
LIN {X -129.2789,Y 11.3864,Z 150,A 172.0348,B 22.3025,C -1.0394,E1 22.1659,E2 275.2441} C_DIS
LIN {X -128.9159,Y 14.9439,Z 150,A 170.3767,B 22.3024,C -1.0412,E1 22.1664,E2 276.9088} C_DIS
LIN {X -128.6092,Y 17.39,Z 150,A 169.0754,B 22.3026,C -1.036,E1 22.1669,E2 278.2328} C_DIS
LIN {X -128.0221,Y 21.2785,Z 150,A 167.4156,B 22.3022,C -1.0447,E1 22.1676,E2 279.8808} C_DIS
LIN {X -127.3659,Y 24.9132,Z 150,A 165.6625,B 22.3022,C -1.0449,E1 22.1685,E2 281.6452} C_DIS
LIN {X -126.4896,Y 29.0312,Z 150,A 163.9301,B 22.3017,C -1.0559,E1 22.1695,E2 283.3598} C_DIS
LIN {X -125.6139,Y 32.6199,Z 150,A 161.5434,B 22.3029,C -1.0303,E1 22.1713,E2 285.8304} C_DIS
LIN {X -124.179,Y 37.7101,Z 150,A 159.8974,B 22.3013,C -1.0656,E1 22.1725,E2 287.3935} C_DIS
LIN {X -123.1189,Y 41.0381,Z 150,A 158.3589,B 22.3011,C -1.0706,E1 22.1738,E2 288.9288} C_DIS
LIN {X -121.8439,Y 44.6873,Z 150,A 156.428,B 22.3012,C -1.0666,E1 22.1757,E2 290.8827} C_DIS
LIN {X -120.2017,Y 48.9295,Z 150,A 154.6538,B 22.3005,C -1.0823,E1 22.1775,E2 292.6265} C_DIS
LIN {X -119.0373,Y 51.6965,Z 150,A 153.3199,B 22.3003,C -1.086,E1 22.1789,E2 293.9591} C_DIS
LIN {X -115.7209,Y 58.7455,Z 150,A 149.7684,B 22.3001,C -1.0916,E1 22.1832,E2 297.5177} C_DIS
LIN {X -113.8831,Y 62.2374,Z 150,A 148.0005,B 22.2999,C -1.0955,E1 22.1855,E2 299.2857} C_DIS
LIN {X -110.6733,Y 67.7811,Z 150,A 145.3276,B 22.2992,C -1.11,E1 22.1893,E2 301.936} C_DIS
LIN {X -108.4699,Y 71.2538,Z 150,A 143.495,B 22.299,C -1.1144,E1 22.192,E2 303.7675} C_DIS
LIN {X -106.4449,Y 74.2451,Z 150,A 141.4692,B 22.2997,C -1.101,E1 22.1953,E2 305.8402} C_DIS
LIN {X -104.5036,Y 76.9537,Z 150,A 140.4421,B 22.2986,C -1.1232,E1 22.1969,E2 306.814} C_DIS
LIN {X -102.5348,Y 79.5579,Z 150,A 138.7229,B 22.299,C -1.1156,E1 22.1999,E2 308.5627} C_DIS
LIN {X -99.9375,Y 82.797,Z 150,A 136.9427,B 22.2986,C -1.1225,E1 22.203,E2 310.334} C_DIS
LIN {X -97.0439,Y 86.1707,Z 150,A 134.9697,B 22.2984,C -1.127,E1 22.2066,E2 312.3052} C_DIS
LIN {X -92.3545,Y 91.1792,Z 150,A 132.0009,B 22.2979,C -1.1369,E1 22.2123,E2 315.2623} C_DIS
LIN {X -89.5062,Y 93.9763,Z 150,A 129.6774,B 22.2989,C -1.1178,E1 22.2171,E2 317.6475} C_DIS
LIN {X -86.2168,Y 97.0032,Z 150,A 127.7513,B 22.2986,C -1.1242,E1 22.2211,E2 319.5653} C_DIS
LIN {X -83.0589,Y 99.7206,Z 150,A 126.2921,B 22.2976,C -1.144,E1 22.2242,E2 320.9784} C_DIS
LIN {X -79.0383,Y 102.9361,Z 150,A 123.8066,B 22.2978,C -1.14,E1 22.2297,E2 323.485} C_DIS
LIN {X -76.4481,Y 104.8745,Z 150,A 122.3946,B 22.2976,C -1.1436,E1 22.2328,E2 324.8932} C_DIS
LIN {X -72.8892,Y 107.378,Z 150,A 120.6469,B 22.2971,C -1.1546,E1 22.2368,E2 326.6184} C_DIS
LIN {X -69.386,Y 109.6743,Z 150,A 118.3045,B 22.2979,C -1.1374,E1 22.2425,E2 329.0149} C_DIS
LIN {X -65.4163,Y 112.0878,Z 150,A 117.0317,B 22.2961,C -1.1738,E1 22.2453,E2 330.1958} C_DIS
LIN {X -60.534,Y 114.7956,Z 150,A 114.5983,B 22.2959,C -1.1793,E1 22.2512,E2 332.6225} C_DIS
LIN {X -56.9406,Y 116.6207,Z 150,A 112.4838,B 22.2964,C -1.1678,E1 22.2566,E2 334.7737} C_DIS
LIN {X -52.4049,Y 118.7282,Z 150,A 110.2502,B 22.2964,C -1.17,E1 22.2623,E2 337.0078} C_DIS
LIN {X -48.3034,Y 120.4541,Z 150,A 108.3644,B 22.296,C -1.1761,E1 22.2671,E2 338.8823} C_DIS
LIN {X -43.1455,Y 122.3973,Z 150,A 105.4764,B 22.2968,C -1.1598,E1 22.2748,E2 341.82} C_DIS
LIN {X -39.3914,Y 123.6556,Z 150,A 104.2159,B 22.2957,C -1.1826,E1 22.278,E2 343.0228} C_DIS
LIN {X -36.341,Y 124.5863,Z 150,A 102.7814,B 22.2957,C -1.183,E1 22.2818,E2 344.459} C_DIS
LIN {X -33.0954,Y 125.4879,Z 150,A 101.3084,B 22.2956,C -1.1851,E1 22.2858,E2 345.929} C_DIS
LIN {X -30.3431,Y 126.1812,Z 150,A 100.0194,B 22.2956,C -1.1847,E1 22.2893,E2 347.2211} C_DIS
LIN {X -27.1671,Y 126.9032,Z 150,A 98.583,B 22.2956,C -1.186,E1 22.2932,E2 348.6561} C_DIS
LIN {X -23.0172,Y 127.721,Z 150,A 96.429,B 22.2961,C -1.175,E1 22.2992,E2 350.8416} C_DIS
LIN {X -16.2106,Y 128.7637,Z 150,A 93.7344,B 22.2952,C -1.1919,E1 22.3066,E2 353.4943} C_DIS
LIN {X -13.4205,Y 129.0835,Z 150,A 91.5908,B 22.2971,C -1.1534,E1 22.3128,E2 355.7409} C_DIS
LIN {X -7.5145,Y 129.5617,Z 150,A 89.8962,B 22.2951,C -1.1944,E1 22.3172,E2 357.328} C_DIS
LIN {X -1.2564,Y 129.7737,Z 150,A 87.1659,B 22.295,C -1.1966,E1 22.3248,E2 360.0529} C_DIS
LIN {X 1.5954,Y 129.77,Z 150,A 85.4066,B 22.2961,C -1.1748,E1 22.3299,E2 361.8695} C_DIS
LIN {X 5.1041,Y 129.6782,Z 150,A 84.248,B 22.2952,C -1.192,E1 22.333,E2 362.9822} C_DIS
LIN {X 11.4701,Y 129.2718,Z 150,A 81.4817,B 22.2952,C -1.1941,E1 22.3407,E2 365.7417} C_DIS
LIN {X 14.6684,Y 128.9488,Z 150,A 79.7447,B 22.2958,C -1.1797,E1 22.3456,E2 367.5152} C_DIS
LIN {X 22.0553,Y 127.8925,Z 150,A 76.7517,B 22.2952,C -1.1921,E1 22.3538,E2 370.4724} C_DIS
LIN {X 24.7789,Y 127.3915,Z 150,A 75.3292,B 22.2957,C -1.1827,E1 22.3577,E2 371.9179} C_DIS
LIN {X 29.1266,Y 126.4678,Z 150,A 73.6027,B 22.2952,C -1.1922,E1 22.3624,E2 373.6167} C_DIS
LIN {X 32.3222,Y 125.6895,Z 150,A 72.131,B 22.2952,C -1.1904,E1 22.3664,E2 375.0905} C_DIS
LIN {X 34.9222,Y 124.9913,Z 150,A 70.8968,B 22.2954,C -1.1876,E1 22.3697,E2 376.33} C_DIS
LIN {X 38.0587,Y 124.0723,Z 150,A 69.4731,B 22.2954,C -1.1873,E1 22.3735,E2 377.7515} C_DIS
LIN {X 41.0824,Y 123.1041,Z 150,A 68.0481,B 22.2956,C -1.1851,E1 22.3773,E2 379.1792} C_DIS
LIN {X 44.1729,Y 122.0293,Z 150,A 66.6201,B 22.2956,C -1.1846,E1 22.381,E2 380.6054} C_DIS
LIN {X 47.951,Y 120.5962,Z 150,A 64.7807,B 22.2958,C -1.1802,E1 22.3859,E2 382.4516} C_DIS
LIN {X 51.7517,Y 119.0134,Z 150,A 63.0191,B 22.2958,C -1.1808,E1 22.3904,E2 384.2069} C_DIS
LIN {X 55.3067,Y 117.4053,Z 150,A 60.9634,B 22.2966,C -1.1636,E1 22.3957,E2 386.302} C_DIS
LIN {X 58.3227,Y 115.9361,Z 150,A 59.7876,B 22.296,C -1.1756,E1 22.3985,E2 387.4426} C_DIS
LIN {X 61.6912,Y 114.1803,Z 150,A 58.0588,B 22.2963,C -1.1709,E1 22.4028,E2 389.178} C_DIS
LIN {X 65.4829,Y 112.0487,Z 150,A 55.8145,B 22.2971,C -1.1534,E1 22.4083,E2 391.4608} C_DIS
LIN {X 68.7494,Y 110.0745,Z 150,A 54.7247,B 22.2959,C -1.1781,E1 22.4108,E2 392.4819} C_DIS
LIN {X 71.0235,Y 108.6215,Z 150,A 52.9463,B 22.2973,C -1.1492,E1 22.4151,E2 394.3294} C_DIS
LIN {X 74.1801,Y 106.4902,Z 150,A 52.0039,B 22.2958,C -1.1804,E1 22.4171,E2 395.1863} C_DIS
LIN {X 78.2138,Y 103.5638,Z 150,A 49.421,B 22.2969,C -1.1588,E1 22.423,E2 397.8155} C_DIS
LIN {X 81.7626,Y 100.7862,Z 150,A 47.4453,B 22.297,C -1.1557,E1 22.4273,E2 399.7908} C_DIS
LIN {X 85.0491,Y 98.0287,Z 150,A 45.5776,B 22.2971,C -1.1533,E1 22.4313,E2 401.6568} C_DIS
LIN {X 91.2188,Y 92.3147,Z 150,A 42.1904,B 22.2968,C -1.1607,E1 22.4381,E2 405.0086} C_DIS
LIN {X 95.6174,Y 87.7505,Z 150,A 39.1358,B 22.2977,C -1.1425,E1 22.4441,E2 408.0959} C_DIS
LIN {X 98.2215,Y 84.8258,Z 150,A 37.3429,B 22.298,C -1.1356,E1 22.4474,E2 409.898} C_DIS
LIN {X 101.0933,Y 81.3819,Z 150,A 35.4067,B 22.2981,C -1.1329,E1 22.4508,E2 411.8309} C_DIS
LIN {X 103.7873,Y 77.9175,Z 150,A 33.4318,B 22.2984,C -1.1264,E1 22.4542,E2 413.8122} C_DIS
LIN {X 106.3576,Y 74.3707,Z 150,A 31.1042,B 22.2996,C -1.1031,E1 22.458,E2 416.1881} C_DIS
LIN {X 108.7664,Y 70.8007,Z 150,A 29.9569,B 22.2981,C -1.1337,E1 22.4596,E2 417.2488} C_DIS
LIN {X 110.2613,Y 68.4494,Z 150,A 28.0337,B 22.2998,C -1.0977,E1 22.4626,E2 419.255} C_DIS
LIN {X 112.3722,Y 64.9257,Z 150,A 26.7136,B 22.2989,C -1.1161,E1 22.4644,E2 420.5193} C_DIS
LIN {X 114.1332,Y 61.7788,Z 150,A 25.0021,B 22.2994,C -1.1061,E1 22.4667,E2 422.2468} C_DIS
LIN {X 116.2045,Y 57.7843,Z 150,A 23.006,B 22.2997,C -1.1002,E1 22.4692,E2 424.2465} C_DIS
LIN {X 118.1475,Y 53.7041,Z 150,A 21.0248,B 22.2999,C -1.0951,E1 22.4716,E2 426.2287} C_DIS
LIN {X 120.803,Y 47.4257,Z 150,A 18.3411,B 22.2996,C -1.102,E1 22.4744,E2 428.8778} C_DIS
LIN {X 122.1546,Y 43.8254,Z 150,A 16.5183,B 22.3001,C -1.091,E1 22.4762,E2 430.7178} C_DIS
LIN {X 123.2402,Y 40.6738,Z 150,A 14.9291,B 22.3006,C -1.081,E1 22.4776,E2 432.323} C_DIS
LIN {X 124.532,Y 36.5264,Z 150,A 13.0893,B 22.3006,C -1.0789,E1 22.4791,E2 434.1564} C_DIS
LIN {X 125.4881,Y 33.0949,Z 150,A 11.4435,B 22.3011,C -1.0706,E1 22.4803,E2 435.8131} C_DIS
LIN {X 126.6067,Y 28.5186,Z 150,A 8.7661,B 22.3026,C -1.0358,E1 22.482,E2 438.5641} C_DIS
LIN {X 127.6893,Y 23.1942,Z 150,A 7.3172,B 22.3009,C -1.0736,E1 22.4827,E2 439.9044} C_DIS
LIN {X 128.1478,Y 20.5191,Z 150,A 5.1003,B 22.3033,C -1.0212,E1 22.4838,E2 442.2438} C_DIS
LIN {X 128.9534,Y 14.6296,Z 150,A 2.891,B 22.3028,C -1.0325,E1 22.4845,E2 444.4085} C_DIS
LIN {X 129.3212,Y 10.8851,Z 150,A 1.692,B 22.302,C -1.0494,E1 22.4847,E2 445.5552} C_DIS
LIN {X 129.5838,Y 7.1338,Z 150,A -0.1278,B 22.3026,C -1.0364,E1 22.4851,E2 447.3968} C_DIS
LIN {X 129.7745,Y 1.1562,Z 150,A -2.9766,B 22.3034,C -1.018,E1 22.4852,E2 450.2747} C_DIS
LIN {X 129.7559,Y -2.4434,Z 150,A -4.1134,B 22.3027,C -1.0346,E1 22.4852,E2 451.3604} C_DIS
LIN {X 129.6394,Y -6.0287,Z 150,A -6.1975,B 22.3039,C -1.0054,E1 22.4849,E2 453.5066} C_DIS
LIN {X 129.3882,Y -10.0774,Z 150,A -7.5596,B 22.3033,C -1.0202,E1 22.4847,E2 454.8208} C_DIS
LIN {X 128.7439,Y -16.3622,Z 150,A -10.2847,B 22.3036,C -1.0143,E1 22.4838,E2 457.5431} C_DIS
LIN {X 128.2623,Y -19.7794,Z 150,A -11.8269,B 22.3038,C -1.0085,E1 22.4832,E2 459.0901} C_DIS
LIN {X 127.5833,Y -23.7756,Z 150,A -13.7993,B 22.3044,C -0.994,E1 22.4822,E2 461.0874} C_DIS
LIN {X 126.8088,Y -27.6042,Z 150,A -15.2901,B 22.3042,C -0.9998,E1 22.4814,E2 462.5532} C_DIS
LIN {X 125.9838,Y -31.1621,Z 150,A -16.9352,B 22.3045,C -0.9931,E1 22.4803,E2 464.2051} C_DIS
LIN {X 124.5547,Y -36.4489,Z 150,A -19.3358,B 22.3047,C -0.9863,E1 22.4785,E2 466.6078} C_DIS
LIN {X 123.6515,Y -39.4042,Z 150,A -20.6627,B 22.3048,C -0.9838,E1 22.4774,E2 467.9326} C_DIS
LIN {X 122.5556,Y -42.691,Z 150,A -22.1643,B 22.305,C -0.9804,E1 22.476,E2 469.4336} C_DIS
LIN {X 121.5104,Y -45.5806,Z 150,A -23.9953,B 22.3061,C -0.9535,E1 22.4742,E2 471.3234} C_DIS
LIN {X 119.957,Y -49.5272,Z 150,A -25.297,B 22.3052,C -0.9751,E1 22.4729,E2 472.5604} C_DIS
LIN {X 118.9505,Y -51.8971,Z 150,A -26.5871,B 22.3057,C -0.9643,E1 22.4714,E2 473.8708} C_DIS
LIN {X 116.1234,Y -57.9487,Z 150,A -29.4086,B 22.3057,C -0.9616,E1 22.4681,E2 476.6822} C_DIS
LIN {X 114.5837,Y -60.9374,Z 150,A -30.8974,B 22.306,C -0.957,E1 22.4661,E2 478.1741} C_DIS
LIN {X 112.5848,Y -64.557,Z 150,A -32.9678,B 22.3066,C -0.94,E1 22.4633,E2 480.2769} C_DIS
LIN {X 110.1665,Y -68.6016,Z 150,A -34.8487,B 22.3065,C -0.9436,E1 22.4606,E2 482.1374} C_DIS
LIN {X 107.7915,Y -72.2766,Z 150,A -36.6832,B 22.3065,C -0.9428,E1 22.4578,E2 483.9636} C_DIS
LIN {X 105.7548,Y -75.2254,Z 150,A -38.4959,B 22.3071,C -0.9275,E1 22.4548,E2 485.8064} C_DIS
LIN {X 100.5932,Y -81.9992,Z 150,A -41.9394,B 22.3069,C -0.9325,E1 22.449,E2 489.2181} C_DIS
LIN {X 98.9939,Y -83.9231,Z 150,A -43.1701,B 22.3073,C -0.9236,E1 22.4467,E2 490.4658} C_DIS
LIN {X 95.014,Y -88.4035,Z 150,A -45.8299,B 22.3076,C -0.9163,E1 22.4417,E2 493.1314} C_DIS
LIN {X 90.4891,Y -93.0304,Z 150,A -48.7011,B 22.3079,C -0.9087,E1 22.4361,E2 496.0087} C_DIS
LIN {X 87.2148,Y -96.1063,Z 150,A -50.5989,B 22.3079,C -0.9081,E1 22.4322,E2 497.8993} C_DIS
LIN {X 83.6134,Y -99.2557,Z 150,A -53.166,B 22.3089,C -0.8819,E1 22.4266,E2 500.5237} C_DIS
LIN {X 80.2686,Y -101.9794,Z 150,A -54.6463,B 22.3083,C -0.8977,E1 22.4235,E2 501.9562} C_DIS
LIN {X 76.5753,Y -104.7815,Z 150,A -56.6986,B 22.3085,C -0.8932,E1 22.4189,E2 504.012} C_DIS
LIN {X 72.9718,Y -107.3219,Z 150,A -58.7327,B 22.3088,C -0.8852,E1 22.4142,E2 506.0592} C_DIS
LIN {X 69.5115,Y -109.5951,Z 150,A -60.4005,B 22.3086,C -0.8892,E1 22.4103,E2 507.7104} C_DIS
LIN {X 62.0349,Y -113.9936,Z 150,A -63.9661,B 22.3084,C -0.8947,E1 22.4018,E2 511.2494} C_DIS
LIN {X 58.4641,Y -115.8642,Z 150,A -65.9268,B 22.3088,C -0.8832,E1 22.3968,E2 513.2339} C_DIS
LIN {X 54.8772,Y -117.6055,Z 150,A -67.6199,B 22.3088,C -0.8836,E1 22.3926,E2 514.921} C_DIS
LIN {X 52.7368,Y -118.5802,Z 150,A -69.1126,B 22.3097,C -0.861,E1 22.3887,E2 516.469} C_DIS
LIN {X 49.259,Y -120.0675,Z 150,A -70.6129,B 22.3095,C -0.8664,E1 22.3848,E2 517.951} C_DIS
LIN {X 45.5487,Y -121.5224,Z 150,A -72.1261,B 22.3091,C -0.8755,E1 22.3809,E2 519.4367} C_DIS
LIN {X 42.479,Y -122.6292,Z 150,A -73.9161,B 22.3098,C -0.8575,E1 22.3761,E2 521.2697} C_DIS
LIN {X 39.1574,Y -123.7304,Z 150,A -75.0104,B 22.3091,C -0.8764,E1 22.3733,E2 522.312} C_DIS
LIN {X 36.3606,Y -124.5805,Z 150,A -76.3686,B 22.3093,C -0.8719,E1 22.3697,E2 523.6796} C_DIS
LIN {X 33.2762,Y -125.4397,Z 150,A -77.8123,B 22.3093,C -0.869,E1 22.3658,E2 525.1281} C_DIS
LIN {X 27.9839,Y -126.7263,Z 150,A -80.3701,B 22.3097,C -0.8597,E1 22.3588,E2 527.7063} C_DIS
LIN {X 23.8264,Y -127.5736,Z 150,A -82.3465,B 22.3099,C -0.8535,E1 22.3533,E2 529.6965} C_DIS
LIN {X 17.9808,Y -128.5273,Z 150,A -84.6378,B 22.3095,C -0.8664,E1 22.3471,E2 531.9512} C_DIS
LIN {X 12.2883,Y -129.1955,Z 150,A -87.2353,B 22.3096,C -0.8619,E1 22.3399,E2 534.5585} C_DIS
LIN {X 8.1698,Y -129.5213,Z 150,A -89.4173,B 22.3103,C -0.8449,E1 22.3337,E2 536.7841} C_DIS
LIN {X 4.4502,Y -129.7037,Z 150,A -90.7708,B 22.3098,C -0.8574,E1 22.33,E2 538.1042} C_DIS
LIN {X 0.9288,Y -129.7622,Z 150,A -92.0578,B 22.3094,C -0.8694,E1 22.3265,E2 539.3595} C_DIS
Enddeposition()
LIN {X 0.9288,Y -129.7622,Z 150,A -92.0578,B 22.3094,C -0.8694,E1 22.3265,E2 539.3595} C_DIS
Startdeposition()
$VEL.CP = VEL_PRINT
LIN {X 3.609,Y -128.7811,Z 150,A -90.2637,B 21.2645,C -0.7319,E1 21.2818,E2 537.8162} C_DIS
LIN {X 10.0855,Y -128.4381,Z 150,A -87.155,B 21.2641,C -0.7427,E1 21.2906,E2 534.6794} C_DIS
Enddeposition()
END
